Yaskawa INFORM job: A_ROOF_SIDE_0617_2_PAINT_35.JBI

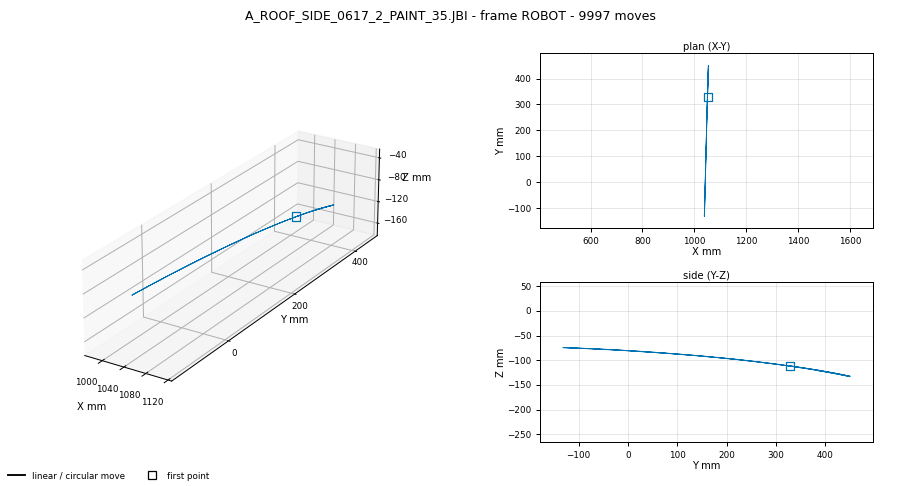
[picture p0: tool path of A_ROOF_SIDE_0617_2_PAINT_35.JBI in frame ROBOT, 9997 of 9997 moves have a stored position in this frame; points joined in program order, loops and branches not executed]
/JOB
//NAME A_ROOF_SIDE_0617_2_PAINT35
//POS
///NPOS 9997,0,0,0,0,0
///TOOL 1
///USER 0
///POSTYPE ROBOT
///RECTAN
///RCONF 1,0,0,0,0,0,0,0,0,0,0,0,0,0,0,0,0,0,0,0,0,0,0,0
C00000=1051.270,329.191,-111.247,172.986,38.897,157.407
C00001=1051.277,329.439,-111.283,172.990,38.901,157.408
C00002=1051.284,329.686,-111.318,172.994,38.904,157.409
C00003=1051.291,329.934,-111.353,172.998,38.908,157.410
C00004=1051.298,330.181,-111.388,173.002,38.912,157.411
C00005=1051.304,330.428,-111.423,173.006,38.916,157.412
C00006=1051.311,330.676,-111.458,173.010,38.920,157.414
C00007=1051.318,330.923,-111.494,173.014,38.924,157.414
C00008=1051.325,331.171,-111.529,173.018,38.928,157.415
C00009=1051.332,331.419,-111.564,173.022,38.933,157.417
C00010=1051.339,331.666,-111.599,173.026,38.936,157.418
C00011=1051.346,331.913,-111.635,173.031,38.940,157.419
C00012=1051.352,332.161,-111.670,173.035,38.944,157.420
C00013=1051.360,332.446,-111.711,173.039,38.949,157.421
C00014=1051.369,332.732,-111.752,173.044,38.953,157.422
C00015=1051.377,333.018,-111.792,173.049,38.958,157.423
C00016=1051.385,333.305,-111.834,173.054,38.963,157.424
C00017=1051.392,333.552,-111.869,173.058,38.967,157.426
C00018=1051.398,333.799,-111.904,173.062,38.971,157.427
C00019=1051.405,334.047,-111.940,173.066,38.975,157.428
C00020=1051.413,334.294,-111.976,173.070,38.979,157.429
C00021=1051.420,334.541,-112.011,173.075,38.983,157.430
C00022=1051.426,334.789,-112.046,173.079,38.988,157.431
C00023=1051.434,335.036,-112.082,173.083,38.991,157.432
C00024=1051.440,335.284,-112.118,173.087,38.996,157.433
C00025=1051.447,335.531,-112.153,173.092,39.000,157.434
C00026=1051.454,335.778,-112.189,173.096,39.003,157.435
C00027=1051.461,336.026,-112.225,173.100,39.008,157.436
C00028=1051.468,336.273,-112.260,173.104,39.012,157.437
C00029=1051.475,336.520,-112.296,173.109,39.016,157.438
C00030=1051.482,336.768,-112.332,173.113,39.021,157.439
C00031=1051.489,337.015,-112.367,173.117,39.024,157.440
C00032=1051.496,337.262,-112.403,173.122,39.029,157.441
C00033=1051.503,337.510,-112.439,173.126,39.033,157.442
C00034=1051.510,337.757,-112.475,173.130,39.037,157.444
C00035=1051.517,338.004,-112.511,173.134,39.041,157.445
C00036=1051.524,338.252,-112.547,173.139,39.045,157.446
C00037=1051.531,338.499,-112.583,173.143,39.050,157.447
C00038=1051.538,338.747,-112.619,173.147,39.054,157.448
C00039=1051.545,338.994,-112.654,173.152,39.058,157.449
C00040=1051.551,339.241,-112.691,173.156,39.062,157.450
C00041=1051.559,339.488,-112.727,173.160,39.067,157.451
C00042=1051.566,339.736,-112.762,173.165,39.071,157.452
C00043=1051.573,339.984,-112.799,173.169,39.075,157.453
C00044=1051.580,340.230,-112.835,173.173,39.079,157.455
C00045=1051.587,340.478,-112.872,173.178,39.084,157.456
C00046=1051.594,340.725,-112.908,173.182,39.088,157.457
C00047=1051.601,340.973,-112.943,173.186,39.092,157.458
C00048=1051.607,341.220,-112.979,173.191,39.096,157.459
C00049=1051.615,341.467,-113.016,173.195,39.101,157.460
C00050=1051.622,341.714,-113.052,173.199,39.105,157.461
C00051=1051.629,341.962,-113.088,173.204,39.109,157.462
C00052=1051.636,342.209,-113.124,173.209,39.114,157.464
C00053=1051.644,342.456,-113.160,173.213,39.117,157.465
C00054=1051.650,342.703,-113.197,173.218,39.122,157.466
C00055=1051.658,342.951,-113.233,173.222,39.126,157.467
C00056=1051.664,343.198,-113.270,173.227,39.131,157.468
C00057=1051.671,343.445,-113.306,173.231,39.135,157.469
C00058=1051.678,343.692,-113.342,173.235,39.139,157.470
C00059=1051.685,343.940,-113.379,173.240,39.144,157.471
C00060=1051.693,344.187,-113.416,173.244,39.148,157.473
C00061=1051.700,344.434,-113.452,173.249,39.152,157.474
C00062=1051.706,344.681,-113.489,173.253,39.157,157.475
C00063=1051.714,344.928,-113.525,173.258,39.162,157.476
C00064=1051.720,345.176,-113.562,173.262,39.166,157.477
C00065=1051.728,345.423,-113.599,173.266,39.170,157.478
C00066=1051.735,345.670,-113.635,173.272,39.175,157.480
C00067=1051.742,345.918,-113.672,173.276,39.179,157.481
C00068=1051.749,346.165,-113.708,173.281,39.183,157.482
C00069=1051.758,346.447,-113.751,173.286,39.189,157.483
C00070=1051.765,346.728,-113.792,173.291,39.194,157.485
C00071=1051.773,347.010,-113.834,173.296,39.199,157.486
C00072=1051.782,347.292,-113.876,173.301,39.204,157.487
C00073=1051.789,347.540,-113.913,173.306,39.209,157.489
C00074=1051.795,347.787,-113.950,173.310,39.213,157.490
C00075=1051.803,348.035,-113.987,173.315,39.218,157.491
C00076=1051.810,348.281,-114.023,173.319,39.222,157.492
C00077=1051.817,348.528,-114.061,173.324,39.227,157.493
C00078=1051.824,348.776,-114.098,173.328,39.231,157.494
C00079=1051.832,349.023,-114.135,173.334,39.236,157.496
C00080=1051.839,349.270,-114.172,173.338,39.240,157.497
C00081=1051.846,349.517,-114.209,173.343,39.245,157.498
C00082=1051.853,349.764,-114.246,173.348,39.249,157.499
C00083=1051.860,350.012,-114.282,173.352,39.254,157.500
C00084=1051.868,350.259,-114.320,173.357,39.259,157.502
C00085=1051.874,350.505,-114.357,173.361,39.263,157.503
C00086=1051.881,350.753,-114.394,173.367,39.268,157.504
C00087=1051.889,351.000,-114.431,173.371,39.272,157.505
C00088=1051.896,351.247,-114.468,173.376,39.277,157.507
C00089=1051.904,351.494,-114.506,173.380,39.281,157.508
C00090=1051.911,351.741,-114.543,173.385,39.286,157.509
C00091=1051.917,351.988,-114.580,173.389,39.291,157.510
C00092=1051.925,352.236,-114.617,173.395,39.296,157.512
C00093=1051.932,352.483,-114.655,173.400,39.300,157.513
C00094=1051.939,352.730,-114.692,173.404,39.305,157.514
C00095=1051.946,352.977,-114.730,173.409,39.310,157.515
C00096=1051.954,353.224,-114.767,173.414,39.315,157.517
C00097=1051.961,353.471,-114.805,173.419,39.319,157.518
C00098=1051.968,353.718,-114.842,173.424,39.324,157.519
C00099=1051.975,353.966,-114.880,173.428,39.329,157.520
C00100=1051.982,354.212,-114.917,173.433,39.333,157.522
C00101=1051.989,354.459,-114.955,173.437,39.338,157.523
C00102=1051.996,354.706,-114.992,173.443,39.343,157.524
C00103=1052.004,354.953,-115.030,173.448,39.348,157.525
C00104=1052.011,355.201,-115.067,173.452,39.352,157.527
C00105=1052.018,355.447,-115.106,173.457,39.357,157.528
C00106=1052.026,355.694,-115.143,173.463,39.362,157.529
C00107=1052.033,355.941,-115.181,173.467,39.366,157.531
C00108=1052.040,356.188,-115.218,173.472,39.371,157.532
C00109=1052.047,356.436,-115.256,173.477,39.376,157.533
C00110=1052.056,356.683,-115.294,173.482,39.381,157.534
C00111=1052.063,356.930,-115.332,173.487,39.386,157.536
C00112=1052.070,357.177,-115.369,173.492,39.391,157.537
C00113=1052.078,357.424,-115.408,173.496,39.396,157.538
C00114=1052.085,357.671,-115.445,173.502,39.401,157.540
C00115=1052.091,357.918,-115.483,173.507,39.405,157.541
C00116=1052.099,358.165,-115.521,173.511,39.410,157.542
C00117=1052.106,358.412,-115.559,173.516,39.415,157.544
C00118=1052.114,358.658,-115.597,173.522,39.420,157.545
C00119=1052.121,358.905,-115.635,173.527,39.425,157.546
C00120=1052.128,359.152,-115.674,173.531,39.430,157.548
C00121=1052.136,359.400,-115.711,173.537,39.435,157.549
C00122=1052.143,359.647,-115.750,173.542,39.440,157.550
C00123=1052.150,359.894,-115.787,173.546,39.445,157.552
C00124=1052.158,360.140,-115.825,173.551,39.450,157.553
C00125=1052.164,360.354,-115.859,173.555,39.454,157.554
C00126=1052.170,360.566,-115.892,173.561,39.458,157.555
C00127=1052.177,360.780,-115.924,173.565,39.463,157.556
C00128=1052.183,360.993,-115.957,173.569,39.467,157.558
C00129=1052.190,361.206,-115.990,173.573,39.471,157.559
C00130=1052.196,361.419,-116.024,173.578,39.476,157.560
C00131=1052.202,361.632,-116.057,173.582,39.480,157.561
C00132=1052.209,361.845,-116.090,173.587,39.485,157.562
C00133=1052.216,362.092,-116.128,173.592,39.489,157.564
C00134=1052.223,362.339,-116.167,173.597,39.495,157.565
C00135=1052.230,362.586,-116.205,173.603,39.500,157.567
C00136=1052.239,362.833,-116.243,173.607,39.505,157.568
C00137=1052.249,363.188,-116.298,173.615,39.512,157.570
C00138=1052.260,363.542,-116.354,173.622,39.520,157.572
C00139=1052.270,363.898,-116.410,173.630,39.527,157.574
C00140=1052.281,364.252,-116.465,173.637,39.534,157.576
C00141=1052.288,364.499,-116.504,173.642,39.539,157.577
C00142=1052.296,364.746,-116.543,173.647,39.545,157.579
C00143=1052.303,364.993,-116.582,173.653,39.550,157.580
C00144=1052.310,365.239,-116.620,173.658,39.555,157.582
C00145=1052.318,365.487,-116.659,173.664,39.560,157.583
C00146=1052.325,365.733,-116.698,173.669,39.566,157.585
C00147=1052.332,365.980,-116.737,173.674,39.571,157.586
C00148=1052.340,366.227,-116.776,173.679,39.576,157.587
C00149=1052.347,366.473,-116.815,173.684,39.581,157.589
C00150=1052.355,366.721,-116.854,173.690,39.587,157.590
C00151=1052.362,366.968,-116.892,173.695,39.592,157.592
C00152=1052.370,367.214,-116.932,173.701,39.597,157.593
C00153=1052.378,367.461,-116.970,173.706,39.603,157.595
C00154=1052.385,367.708,-117.009,173.711,39.608,157.596
C00155=1052.392,367.955,-117.049,173.717,39.613,157.598
C00156=1052.400,368.201,-117.087,173.722,39.619,157.599
C00157=1052.408,368.448,-117.127,173.728,39.624,157.601
C00158=1052.415,368.695,-117.165,173.732,39.630,157.602
C00159=1052.423,368.942,-117.205,173.738,39.635,157.603
C00160=1052.430,369.188,-117.244,173.743,39.640,157.605
C00161=1052.438,369.435,-117.284,173.749,39.646,157.606
C00162=1052.445,369.682,-117.323,173.754,39.651,157.608
C00163=1052.453,369.928,-117.362,173.760,39.656,157.609
C00164=1052.461,370.176,-117.401,173.765,39.662,157.611
C00165=1052.468,370.422,-117.440,173.770,39.667,157.612
C00166=1052.476,370.669,-117.480,173.776,39.673,157.614
C00167=1052.484,370.916,-117.519,173.782,39.678,157.615
C00168=1052.491,371.162,-117.559,173.787,39.684,157.617
C00169=1052.499,371.409,-117.598,173.792,39.689,157.618
C00170=1052.507,371.657,-117.637,173.798,39.695,157.620
C00171=1052.514,371.903,-117.677,173.804,39.700,157.621
C00172=1052.522,372.150,-117.717,173.809,39.705,157.623
C00173=1052.529,372.397,-117.756,173.816,39.711,157.625
C00174=1052.536,372.643,-117.796,173.821,39.716,157.626
C00175=1052.544,372.890,-117.836,173.827,39.722,157.628
C00176=1052.553,373.136,-117.875,173.832,39.728,157.629
C00177=1052.560,373.382,-117.915,173.838,39.734,157.631
C00178=1052.567,373.629,-117.955,173.843,39.739,157.632
C00179=1052.575,373.876,-117.995,173.849,39.745,157.634
C00180=1052.582,374.122,-118.034,173.855,39.751,157.635
C00181=1052.592,374.429,-118.084,173.861,39.758,157.637
C00182=1052.602,374.735,-118.133,173.868,39.765,157.639
C00183=1052.611,375.040,-118.183,173.875,39.772,157.641
C00184=1052.620,375.347,-118.233,173.882,39.779,157.643
C00185=1052.628,375.594,-118.272,173.888,39.785,157.645
C00186=1052.636,375.840,-118.313,173.895,39.791,157.647
C00187=1052.644,376.087,-118.353,173.900,39.796,157.648
C00188=1052.651,376.333,-118.392,173.906,39.802,157.650
C00189=1052.659,376.580,-118.432,173.911,39.808,157.651
C00190=1052.667,376.826,-118.473,173.917,39.813,157.653
C00191=1052.675,377.073,-118.513,173.923,39.819,157.655
C00192=1052.683,377.320,-118.553,173.929,39.825,157.656
C00193=1052.690,377.566,-118.593,173.935,39.831,157.658
C00194=1052.698,377.813,-118.633,173.941,39.837,157.659
C00195=1052.706,378.060,-118.674,173.946,39.843,157.661
C00196=1052.714,378.307,-118.714,173.952,39.848,157.663
C00197=1052.722,378.553,-118.754,173.959,39.854,157.664
C00198=1052.730,378.800,-118.794,173.964,39.860,157.666
C00199=1052.738,379.046,-118.835,173.970,39.866,157.668
C00200=1052.746,379.292,-118.875,173.976,39.872,157.669
C00201=1052.753,379.539,-118.915,173.981,39.878,157.671
C00202=1052.761,379.786,-118.956,173.988,39.884,157.673
C00203=1052.769,380.032,-118.996,173.994,39.890,157.674
C00204=1052.776,380.279,-119.037,173.999,39.896,157.676
C00205=1052.784,380.525,-119.078,174.005,39.902,157.678
C00206=1052.792,380.772,-119.118,174.012,39.908,157.679
C00207=1052.800,381.018,-119.160,174.018,39.914,157.681
C00208=1052.808,381.264,-119.200,174.023,39.920,157.683
C00209=1052.815,381.511,-119.240,174.030,39.926,157.685
C00210=1052.823,381.758,-119.281,174.036,39.932,157.686
C00211=1052.831,382.004,-119.322,174.042,39.938,157.688
C00212=1052.839,382.251,-119.363,174.047,39.944,157.690
C00213=1052.846,382.497,-119.404,174.054,39.951,157.692
C00214=1052.854,382.743,-119.445,174.060,39.957,157.693
C00215=1052.862,382.990,-119.485,174.066,39.963,157.695
C00216=1052.870,383.236,-119.527,174.072,39.969,157.697
C00217=1052.878,383.483,-119.568,174.078,39.975,157.699
C00218=1052.886,383.729,-119.609,174.084,39.981,157.700
C00219=1052.894,383.976,-119.650,174.091,39.988,157.702
C00220=1052.902,384.222,-119.691,174.097,39.994,157.704
C00221=1052.910,384.469,-119.732,174.104,40.000,157.706
C00222=1052.918,384.715,-119.774,174.109,40.007,157.707
C00223=1052.926,384.961,-119.814,174.115,40.013,157.709
C00224=1052.933,385.208,-119.855,174.122,40.019,157.711
C00225=1052.942,385.454,-119.897,174.128,40.025,157.713
C00226=1052.950,385.700,-119.938,174.135,40.031,157.714
C00227=1052.957,385.947,-119.979,174.140,40.038,157.716
C00228=1052.966,386.193,-120.021,174.147,40.044,157.718
C00229=1052.974,386.440,-120.062,174.153,40.051,157.720
C00230=1052.982,386.686,-120.103,174.159,40.057,157.722
C00231=1052.991,386.933,-120.144,174.166,40.063,157.724
C00232=1052.998,387.178,-120.186,174.172,40.070,157.725
C00233=1053.006,387.425,-120.227,174.179,40.076,157.727
C00234=1053.014,387.671,-120.269,174.185,40.082,157.729
C00235=1053.022,387.918,-120.310,174.192,40.089,157.731
C00236=1053.031,388.164,-120.352,174.198,40.096,157.733
C00237=1053.042,388.502,-120.409,174.207,40.104,157.735
C00238=1053.054,388.841,-120.466,174.216,40.113,157.738
C00239=1053.064,389.179,-120.523,174.224,40.122,157.741
C00240=1053.076,389.518,-120.580,174.233,40.131,157.743
C00241=1053.084,389.763,-120.622,174.240,40.137,157.745
C00242=1053.092,390.010,-120.664,174.246,40.144,157.747
C00243=1053.101,390.256,-120.706,174.253,40.151,157.749
C00244=1053.109,390.503,-120.748,174.260,40.157,157.751
C00245=1053.116,390.748,-120.790,174.266,40.164,157.753
C00246=1053.125,390.995,-120.832,174.273,40.171,157.755
C00247=1053.133,391.241,-120.874,174.279,40.178,157.757
C00248=1053.141,391.487,-120.916,174.286,40.184,157.758
C00249=1053.149,391.733,-120.957,174.293,40.191,157.760
C00250=1053.158,391.980,-120.999,174.299,40.198,157.762
C00251=1053.166,392.226,-121.043,174.306,40.204,157.764
C00252=1053.174,392.472,-121.084,174.313,40.211,157.766
C00253=1053.183,392.718,-121.126,174.319,40.218,157.768
C00254=1053.191,392.965,-121.168,174.326,40.225,157.770
C00255=1053.199,393.210,-121.211,174.333,40.232,157.772
C00256=1053.207,393.457,-121.253,174.340,40.238,157.774
C00257=1053.215,393.704,-121.296,174.347,40.245,157.776
C00258=1053.223,393.949,-121.338,174.354,40.252,157.778
C00259=1053.232,394.195,-121.380,174.360,40.259,157.780
C00260=1053.240,394.441,-121.423,174.367,40.266,157.782
C00261=1053.248,394.687,-121.465,174.374,40.273,157.784
C00262=1053.256,394.933,-121.508,174.380,40.280,157.786
C00263=1053.265,395.180,-121.550,174.387,40.287,157.788
C00264=1053.273,395.426,-121.593,174.394,40.294,157.790
C00265=1053.282,395.672,-121.636,174.402,40.301,157.792
C00266=1053.290,395.918,-121.678,174.408,40.308,157.794
C00267=1053.299,396.164,-121.721,174.415,40.315,157.796
C00268=1053.307,396.410,-121.764,174.422,40.322,157.798
C00269=1053.315,396.657,-121.806,174.429,40.329,157.801
C00270=1053.324,396.903,-121.849,174.436,40.336,157.803
C00271=1053.332,397.149,-121.892,174.443,40.343,157.805
C00272=1053.341,397.395,-121.935,174.450,40.351,157.807
C00273=1053.349,397.641,-121.978,174.457,40.358,157.809
C00274=1053.358,397.887,-122.021,174.464,40.364,157.811
C00275=1053.365,398.134,-122.064,174.472,40.372,157.813
C00276=1053.374,398.380,-122.107,174.479,40.379,157.815
C00277=1053.382,398.626,-122.150,174.485,40.386,157.817
C00278=1053.391,398.871,-122.194,174.492,40.394,157.820
C00279=1053.399,399.117,-122.237,174.500,40.401,157.822
C00280=1053.408,399.364,-122.280,174.507,40.408,157.824
C00281=1053.417,399.610,-122.323,174.514,40.415,157.826
C00282=1053.425,399.856,-122.366,174.522,40.423,157.828
C00283=1053.434,400.102,-122.409,174.529,40.430,157.830
C00284=1053.442,400.348,-122.452,174.536,40.438,157.833
C00285=1053.450,400.593,-122.497,174.544,40.445,157.835
C00286=1053.459,400.840,-122.540,174.551,40.452,157.837
C00287=1053.468,401.086,-122.583,174.558,40.459,157.839
C00288=1053.476,401.332,-122.627,174.566,40.467,157.841
C00289=1053.485,401.578,-122.670,174.573,40.474,157.843
C00290=1053.493,401.824,-122.713,174.581,40.482,157.846
C00291=1053.502,402.070,-122.757,174.588,40.489,157.848
C00292=1053.511,402.316,-122.800,174.595,40.497,157.850
C00293=1053.523,402.672,-122.864,174.606,40.508,157.853
C00294=1053.535,403.029,-122.927,174.616,40.519,157.857
C00295=1053.548,403.385,-122.991,174.627,40.530,157.860
C00296=1053.561,403.741,-123.054,174.638,40.541,157.863
C00297=1053.569,403.987,-123.097,174.646,40.549,157.866
C00298=1053.578,404.234,-123.142,174.653,40.557,157.868
C00299=1053.587,404.479,-123.186,174.661,40.564,157.870
C00300=1053.595,404.725,-123.231,174.668,40.572,157.873
C00301=1053.604,404.971,-123.274,174.676,40.580,157.875
C00302=1053.613,405.216,-123.318,174.683,40.588,157.877
C00303=1053.621,405.463,-123.363,174.692,40.595,157.880
C00304=1053.630,405.708,-123.407,174.699,40.603,157.882
C00305=1053.639,405.955,-123.451,174.707,40.611,157.884
C00306=1053.647,406.200,-123.496,174.715,40.619,157.887
C00307=1053.656,406.446,-123.540,174.722,40.627,157.889
C00308=1053.664,406.692,-123.584,174.730,40.634,157.891
C00309=1053.674,406.938,-123.628,174.738,40.643,157.894
C00310=1053.682,407.184,-123.672,174.746,40.650,157.896
C00311=1053.691,407.431,-123.717,174.754,40.659,157.899
C00312=1053.700,407.675,-123.762,174.761,40.666,157.901
C00313=1053.708,407.922,-123.806,174.770,40.674,157.903
C00314=1053.718,408.168,-123.850,174.778,40.683,157.906
C00315=1053.726,408.413,-123.895,174.785,40.690,157.908
C00316=1053.735,408.660,-123.940,174.793,40.699,157.911
C00317=1053.745,408.905,-123.985,174.802,40.707,157.913
C00318=1053.753,409.151,-124.029,174.809,40.715,157.916
C00319=1053.762,409.397,-124.075,174.817,40.723,157.918
C00320=1053.771,409.643,-124.119,174.826,40.731,157.921
C00321=1053.779,409.888,-124.164,174.833,40.740,157.923
C00322=1053.789,410.134,-124.208,174.841,40.748,157.926
C00323=1053.798,410.380,-124.253,174.850,40.756,157.928
C00324=1053.807,410.626,-124.299,174.858,40.764,157.931
C00325=1053.816,410.872,-124.343,174.866,40.772,157.933
C00326=1053.825,411.118,-124.388,174.874,40.781,157.936
C00327=1053.834,411.363,-124.433,174.883,40.789,157.938
C00328=1053.843,411.608,-124.478,174.891,40.797,157.941
C00329=1053.852,411.854,-124.524,174.900,40.805,157.943
C00330=1053.861,412.101,-124.568,174.907,40.814,157.946
C00331=1053.871,412.346,-124.613,174.915,40.822,157.948
C00332=1053.880,412.592,-124.659,174.924,40.831,157.951
C00333=1053.889,412.838,-124.704,174.933,40.839,157.954
C00334=1053.898,413.083,-124.749,174.941,40.847,157.956
C00335=1053.907,413.329,-124.794,174.950,40.856,157.959
C00336=1053.916,413.575,-124.840,174.958,40.865,157.961
C00337=1053.926,413.820,-124.886,174.967,40.873,157.964
C00338=1053.935,414.066,-124.931,174.975,40.882,157.967
C00339=1053.944,414.312,-124.977,174.984,40.891,157.969
C00340=1053.952,414.558,-125.022,174.992,40.899,157.972
C00341=1053.962,414.803,-125.068,175.000,40.908,157.975
C00342=1053.971,415.049,-125.114,175.009,40.917,157.977
C00343=1053.981,415.294,-125.160,175.017,40.925,157.980
C00344=1053.990,415.540,-125.206,175.026,40.934,157.983
C00345=1053.999,415.785,-125.252,175.035,40.942,157.985
C00346=1054.008,416.031,-125.297,175.044,40.952,157.988
C00347=1054.017,416.276,-125.343,175.053,40.960,157.991
C00348=1054.026,416.522,-125.389,175.062,40.969,157.994
C00349=1054.040,416.885,-125.458,175.074,40.982,157.998
C00350=1054.054,417.248,-125.525,175.088,40.995,158.002
C00351=1054.068,417.610,-125.593,175.100,41.008,158.006
C00352=1054.081,417.972,-125.661,175.114,41.021,158.010
C00353=1054.091,418.218,-125.708,175.123,41.031,158.013
C00354=1054.101,418.463,-125.754,175.132,41.040,158.016
C00355=1054.110,418.709,-125.800,175.141,41.049,158.019
C00356=1054.120,418.955,-125.846,175.150,41.058,158.021
C00357=1054.129,419.200,-125.892,175.159,41.067,158.024
C00358=1054.139,419.446,-125.939,175.168,41.076,158.027
C00359=1054.148,419.691,-125.985,175.177,41.085,158.030
C00360=1054.157,419.937,-126.032,175.187,41.094,158.033
C00361=1054.167,420.182,-126.079,175.196,41.104,158.036
C00362=1054.177,420.428,-126.126,175.205,41.113,158.039
C00363=1054.185,420.673,-126.172,175.215,41.122,158.042
C00364=1054.196,420.918,-126.219,175.224,41.131,158.045
C00365=1054.205,421.164,-126.266,175.233,41.141,158.048
C00366=1054.214,421.409,-126.313,175.243,41.150,158.050
C00367=1054.224,421.654,-126.360,175.252,41.160,158.053
C00368=1054.234,421.900,-126.407,175.261,41.169,158.056
C00369=1054.243,422.146,-126.454,175.271,41.178,158.059
C00370=1054.252,422.390,-126.501,175.280,41.188,158.062
C00371=1054.263,422.636,-126.548,175.290,41.197,158.065
C00372=1054.272,422.882,-126.595,175.299,41.207,158.068
C00373=1054.281,423.126,-126.642,175.308,41.216,158.071
C00374=1054.292,423.372,-126.689,175.319,41.226,158.074
C00375=1054.301,423.617,-126.737,175.328,41.235,158.078
C00376=1054.311,423.863,-126.783,175.338,41.246,158.081
C00377=1054.321,424.108,-126.830,175.347,41.255,158.084
C00378=1054.330,424.353,-126.878,175.357,41.265,158.087
C00379=1054.340,424.599,-126.925,175.368,41.274,158.090
C00380=1054.350,424.844,-126.973,175.377,41.284,158.093
C00381=1054.360,425.090,-127.020,175.387,41.294,158.096
C00382=1054.370,425.334,-127.068,175.397,41.303,158.099
C00383=1054.380,425.580,-127.116,175.407,41.313,158.103
C00384=1054.390,425.825,-127.163,175.417,41.324,158.106
C00385=1054.399,426.071,-127.211,175.427,41.333,158.109
C00386=1054.410,426.316,-127.258,175.437,41.343,158.112
C00387=1054.419,426.561,-127.307,175.447,41.353,158.115
C00388=1054.429,426.807,-127.355,175.457,41.363,158.118
C00389=1054.439,427.051,-127.403,175.467,41.373,158.122
C00390=1054.449,427.297,-127.450,175.477,41.383,158.125
C00391=1054.459,427.542,-127.498,175.488,41.393,158.128
C00392=1054.469,427.786,-127.547,175.497,41.403,158.131
C00393=1054.478,428.032,-127.595,175.508,41.414,158.135
C00394=1054.489,428.277,-127.643,175.518,41.424,158.138
C00395=1054.499,428.522,-127.691,175.529,41.433,158.141
C00396=1054.508,428.767,-127.739,175.539,41.444,158.145
C00397=1054.519,429.013,-127.787,175.550,41.454,158.148
C00398=1054.529,429.258,-127.836,175.560,41.464,158.151
C00399=1054.539,429.503,-127.884,175.570,41.475,158.155
C00400=1054.549,429.747,-127.932,175.581,41.485,158.158
C00401=1054.560,429.993,-127.981,175.591,41.496,158.161
C00402=1054.569,430.238,-128.030,175.602,41.506,158.165
C00403=1054.579,430.483,-128.078,175.613,41.516,158.168
C00404=1054.589,430.727,-128.127,175.623,41.527,158.172
C00405=1054.606,431.112,-128.204,175.641,41.543,158.177
C00406=1054.621,431.497,-128.280,175.657,41.560,158.183
C00407=1054.638,431.882,-128.357,175.674,41.577,158.188
C00408=1054.653,432.266,-128.434,175.692,41.593,158.194
C00409=1054.664,432.511,-128.483,175.703,41.604,158.197
C00410=1054.675,432.755,-128.532,175.713,41.615,158.201
C00411=1054.685,433.001,-128.581,175.724,41.625,158.204
C00412=1054.695,433.245,-128.630,175.735,41.636,158.208
C00413=1054.706,433.491,-128.680,175.747,41.647,158.211
C00414=1054.715,433.735,-128.728,175.758,41.658,158.215
C00415=1054.726,433.981,-128.778,175.769,41.669,158.219
C00416=1054.736,434.225,-128.827,175.780,41.680,158.222
C00417=1054.747,434.470,-128.877,175.792,41.691,158.226
C00418=1054.757,434.715,-128.926,175.803,41.702,158.230
C00419=1054.768,434.960,-128.976,175.814,41.713,158.233
C00420=1054.778,435.204,-129.025,175.826,41.724,158.237
C00421=1054.789,435.449,-129.075,175.837,41.735,158.241
C00422=1054.800,435.694,-129.125,175.849,41.746,158.244
C00423=1054.810,435.939,-129.175,175.860,41.757,158.248
C00424=1054.821,436.183,-129.224,175.873,41.768,158.252
C00425=1054.831,436.428,-129.273,175.884,41.780,158.256
C00426=1054.842,436.673,-129.324,175.896,41.791,158.260
C00427=1054.853,436.918,-129.373,175.907,41.802,158.263
C00428=1054.864,437.163,-129.423,175.919,41.814,158.267
C00429=1054.874,437.407,-129.473,175.931,41.825,158.271
C00430=1054.885,437.652,-129.524,175.943,41.836,158.275
C00431=1054.896,437.897,-129.573,175.954,41.848,158.279
C00432=1054.907,438.141,-129.624,175.967,41.859,158.283
C00433=1054.917,438.386,-129.675,175.979,41.870,158.286
C00434=1054.928,438.630,-129.725,175.990,41.882,158.290
C00435=1054.939,438.875,-129.775,176.003,41.894,158.294
C00436=1054.950,439.120,-129.825,176.015,41.905,158.298
C00437=1054.961,439.364,-129.875,176.028,41.917,158.302
C00438=1054.972,439.609,-129.927,176.039,41.929,158.306
C00439=1054.983,439.854,-129.977,176.052,41.940,158.310
C00440=1054.994,440.098,-130.028,176.064,41.953,158.314
C00441=1055.004,440.343,-130.079,176.077,41.964,158.318
C00442=1055.015,440.587,-130.129,176.089,41.976,158.322
C00443=1055.027,440.832,-130.180,176.102,41.988,158.326
C00444=1055.037,441.076,-130.231,176.114,42.000,158.331
C00445=1055.048,441.321,-130.282,176.126,42.011,158.335
C00446=1055.060,441.565,-130.333,176.140,42.023,158.339
C00447=1055.070,441.810,-130.384,176.152,42.036,158.343
C00448=1055.082,442.054,-130.435,176.165,42.048,158.347
C00449=1055.094,442.298,-130.486,176.178,42.060,158.351
C00450=1055.104,442.543,-130.537,176.191,42.072,158.355
C00451=1055.116,442.788,-130.589,176.203,42.084,158.360
C00452=1055.126,443.032,-130.640,176.216,42.096,158.364
C00453=1055.138,443.276,-130.692,176.229,42.109,158.368
C00454=1055.149,443.520,-130.743,176.242,42.121,158.372
C00455=1055.161,443.765,-130.795,176.256,42.133,158.377
C00456=1055.171,444.009,-130.846,176.269,42.146,158.381
C00457=1055.183,444.254,-130.898,176.282,42.158,158.385
C00458=1055.194,444.498,-130.949,176.295,42.170,158.390
C00459=1055.205,444.742,-131.001,176.309,42.183,158.394
C00460=1055.217,444.986,-131.054,176.322,42.196,158.399
C00461=1055.232,445.308,-131.121,176.339,42.212,158.404
C00462=1055.247,445.629,-131.189,176.357,42.229,158.410
C00463=1055.262,445.950,-131.257,176.376,42.245,158.416
C00464=1055.278,446.272,-131.326,176.393,42.262,158.422
C00465=1055.289,446.514,-131.378,176.406,42.275,158.426
C00466=1055.301,446.757,-131.430,176.421,42.287,158.431
C00467=1055.314,447.002,-131.481,176.434,42.300,158.435
C00468=1055.327,447.245,-131.532,176.449,42.312,158.440
C00469=1055.341,447.488,-131.582,176.462,42.324,158.444
C00470=1055.356,447.733,-131.632,176.476,42.336,158.448
C00471=1055.373,447.977,-131.681,176.491,42.348,158.453
C00472=1055.389,448.221,-131.729,176.505,42.359,158.457
C00473=1055.406,448.466,-131.777,176.519,42.371,158.461
C00474=1055.425,448.711,-131.824,176.533,42.382,158.465
C00475=1055.444,448.955,-131.870,176.548,42.393,158.469
C00476=1055.463,449.200,-131.917,176.562,42.404,158.473
C00477=1055.484,449.446,-131.962,176.577,42.414,158.477
C00478=1055.506,449.691,-132.007,176.592,42.425,158.481
C00479=1055.527,449.936,-132.051,176.606,42.435,158.485
C00480=1055.550,450.181,-132.095,176.621,42.445,158.489
C00481=1055.229,450.200,-132.384,176.619,42.547,158.518
C00482=1055.205,449.955,-132.340,176.604,42.538,158.514
C00483=1055.183,449.709,-132.297,176.589,42.527,158.510
C00484=1055.161,449.464,-132.252,176.574,42.517,158.506
C00485=1055.141,449.219,-132.206,176.559,42.506,158.502
C00486=1055.121,448.973,-132.160,176.545,42.496,158.498
C00487=1055.101,448.729,-132.114,176.530,42.485,158.494
C00488=1055.083,448.485,-132.066,176.516,42.474,158.490
C00489=1055.066,448.240,-132.018,176.502,42.462,158.486
C00490=1055.048,447.995,-131.971,176.488,42.451,158.482
C00491=1055.032,447.752,-131.922,176.474,42.439,158.477
C00492=1055.018,447.507,-131.872,176.459,42.428,158.473
C00493=1055.003,447.264,-131.823,176.445,42.415,158.469
C00494=1054.985,446.951,-131.757,176.427,42.400,158.463
C00495=1054.970,446.639,-131.691,176.409,42.384,158.457
C00496=1054.954,446.328,-131.625,176.392,42.368,158.451
C00497=1054.939,446.017,-131.558,176.374,42.352,158.446
C00498=1054.928,445.783,-131.509,176.360,42.340,158.441
C00499=1054.917,445.548,-131.459,176.348,42.328,158.437
C00500=1054.906,445.315,-131.409,176.335,42.316,158.433
C00501=1054.895,445.081,-131.359,176.322,42.303,158.429
C00502=1054.884,444.837,-131.307,176.308,42.291,158.424
C00503=1054.873,444.592,-131.255,176.295,42.279,158.420
C00504=1054.860,444.348,-131.203,176.281,42.266,158.415
C00505=1054.849,444.104,-131.152,176.268,42.254,158.411
C00506=1054.838,443.859,-131.100,176.255,42.242,158.407
C00507=1054.826,443.615,-131.049,176.242,42.229,158.403
C00508=1054.816,443.371,-130.997,176.228,42.217,158.398
C00509=1054.804,443.126,-130.946,176.215,42.205,158.394
C00510=1054.793,442.882,-130.894,176.202,42.193,158.390
C00511=1054.781,442.638,-130.843,176.190,42.180,158.385
C00512=1054.771,442.393,-130.791,176.177,42.168,158.381
C00513=1054.759,442.148,-130.740,176.163,42.156,158.377
C00514=1054.748,441.905,-130.689,176.150,42.144,158.373
C00515=1054.737,441.660,-130.637,176.137,42.132,158.369
C00516=1054.726,441.415,-130.587,176.125,42.121,158.365
C00517=1054.714,441.171,-130.536,176.112,42.109,158.360
C00518=1054.704,440.926,-130.485,176.099,42.097,158.356
C00519=1054.693,440.682,-130.434,176.087,42.085,158.352
C00520=1054.681,440.438,-130.383,176.074,42.073,158.348
C00521=1054.671,440.193,-130.333,176.062,42.061,158.344
C00522=1054.660,439.948,-130.282,176.050,42.050,158.340
C00523=1054.648,439.704,-130.231,176.038,42.037,158.336
C00524=1054.638,439.459,-130.180,176.025,42.026,158.332
C00525=1054.627,439.215,-130.130,176.013,42.014,158.328
C00526=1054.616,438.971,-130.079,176.000,42.003,158.324
C00527=1054.605,438.726,-130.029,175.989,41.992,158.320
C00528=1054.594,438.482,-129.979,175.976,41.980,158.316
C00529=1054.584,438.236,-129.928,175.964,41.968,158.312
C00530=1054.573,437.991,-129.878,175.951,41.957,158.308
C00531=1054.562,437.747,-129.827,175.940,41.945,158.304
C00532=1054.551,437.502,-129.777,175.928,41.934,158.301
C00533=1054.541,437.258,-129.728,175.916,41.923,158.297
C00534=1054.530,437.014,-129.677,175.904,41.911,158.293
C00535=1054.519,436.768,-129.628,175.892,41.900,158.289
C00536=1054.508,436.524,-129.578,175.881,41.889,158.285
C00537=1054.497,436.279,-129.528,175.869,41.878,158.281
C00538=1054.487,436.034,-129.478,175.857,41.867,158.278
C00539=1054.476,435.790,-129.428,175.845,41.856,158.274
C00540=1054.465,435.544,-129.378,175.834,41.845,158.270
C00541=1054.454,435.299,-129.329,175.822,41.834,158.267
C00542=1054.444,435.054,-129.279,175.811,41.823,158.263
C00543=1054.434,434.810,-129.230,175.799,41.812,158.259
C00544=1054.423,434.565,-129.180,175.788,41.800,158.255
C00545=1054.412,434.320,-129.131,175.777,41.790,158.252
C00546=1054.402,434.076,-129.081,175.765,41.779,158.248
C00547=1054.392,433.830,-129.032,175.754,41.768,158.245
C00548=1054.381,433.585,-128.982,175.743,41.757,158.241
C00549=1054.371,433.341,-128.933,175.732,41.747,158.237
C00550=1054.360,433.096,-128.883,175.720,41.736,158.234
C00551=1054.350,432.851,-128.835,175.709,41.725,158.230
C00552=1054.339,432.606,-128.786,175.698,41.714,158.227
C00553=1054.329,432.362,-128.737,175.686,41.703,158.223
C00554=1054.312,431.974,-128.660,175.669,41.687,158.217
C00555=1054.296,431.588,-128.582,175.652,41.670,158.212
C00556=1054.281,431.202,-128.504,175.635,41.654,158.206
C00557=1054.265,430.815,-128.428,175.617,41.637,158.201
C00558=1054.254,430.569,-128.379,175.607,41.626,158.197
C00559=1054.244,430.325,-128.330,175.596,41.616,158.194
C00560=1054.234,430.080,-128.281,175.585,41.606,158.191
C00561=1054.224,429.835,-128.233,175.575,41.595,158.187
C00562=1054.214,429.589,-128.184,175.564,41.585,158.184
C00563=1054.203,429.345,-128.136,175.553,41.575,158.180
C00564=1054.194,429.100,-128.088,175.544,41.565,158.177
C00565=1054.184,428.855,-128.039,175.533,41.554,158.174
C00566=1054.173,428.609,-127.991,175.522,41.544,158.170
C00567=1054.163,428.364,-127.943,175.512,41.534,158.167
C00568=1054.153,428.119,-127.894,175.501,41.524,158.164
C00569=1054.143,427.874,-127.846,175.491,41.514,158.160
C00570=1054.133,427.629,-127.798,175.480,41.504,158.157
C00571=1054.123,427.384,-127.751,175.471,41.494,158.154
C00572=1054.113,427.139,-127.702,175.460,41.484,158.151
C00573=1054.104,426.893,-127.654,175.450,41.474,158.147
C00574=1054.093,426.649,-127.606,175.440,41.464,158.144
C00575=1054.084,426.403,-127.559,175.430,41.454,158.141
C00576=1054.073,426.158,-127.511,175.420,41.444,158.138
C00577=1054.064,425.913,-127.463,175.409,41.434,158.135
C00578=1054.054,425.668,-127.416,175.399,41.424,158.131
C00579=1054.044,425.423,-127.367,175.390,41.415,158.128
C00580=1054.034,425.177,-127.320,175.379,41.405,158.125
C00581=1054.024,424.932,-127.272,175.369,41.395,158.122
C00582=1054.014,424.686,-127.225,175.360,41.385,158.119
C00583=1054.004,424.441,-127.178,175.349,41.376,158.116
C00584=1053.994,424.196,-127.130,175.340,41.366,158.113
C00585=1053.984,423.950,-127.083,175.330,41.356,158.109
C00586=1053.975,423.705,-127.035,175.321,41.347,158.106
C00587=1053.965,423.459,-126.988,175.311,41.337,158.103
C00588=1053.955,423.215,-126.941,175.300,41.328,158.100
C00589=1053.946,422.969,-126.894,175.291,41.318,158.097
C00590=1053.936,422.723,-126.847,175.281,41.309,158.094
C00591=1053.926,422.479,-126.800,175.272,41.299,158.091
C00592=1053.917,422.233,-126.752,175.262,41.290,158.088
C00593=1053.907,421.987,-126.705,175.253,41.281,158.085
C00594=1053.897,421.743,-126.658,175.244,41.271,158.082
C00595=1053.888,421.496,-126.611,175.234,41.261,158.079
C00596=1053.878,421.251,-126.564,175.225,41.252,158.076
C00597=1053.869,421.006,-126.518,175.215,41.243,158.073
C00598=1053.859,420.760,-126.470,175.205,41.234,158.070
C00599=1053.850,420.515,-126.424,175.196,41.224,158.067
C00600=1053.840,420.270,-126.377,175.187,41.215,158.064
C00601=1053.830,420.025,-126.331,175.178,41.206,158.062
C00602=1053.821,419.778,-126.284,175.169,41.197,158.059
C00603=1053.812,419.533,-126.238,175.159,41.188,158.056
C00604=1053.802,419.287,-126.191,175.150,41.179,158.053
C00605=1053.792,419.043,-126.144,175.141,41.169,158.050
C00606=1053.783,418.797,-126.098,175.132,41.160,158.047
C00607=1053.773,418.552,-126.052,175.122,41.151,158.044
C00608=1053.763,418.306,-126.005,175.113,41.143,158.042
C00609=1053.754,418.061,-125.959,175.104,41.134,158.039
C00610=1053.741,417.696,-125.891,175.091,41.121,158.035
C00611=1053.726,417.331,-125.822,175.078,41.107,158.030
C00612=1053.713,416.966,-125.754,175.064,41.094,158.026
C00613=1053.698,416.602,-125.685,175.052,41.081,158.022
C00614=1053.689,416.356,-125.640,175.042,41.072,158.019
C00615=1053.680,416.111,-125.593,175.033,41.063,158.017
C00616=1053.671,415.866,-125.547,175.025,41.055,158.014
C00617=1053.662,415.620,-125.502,175.016,41.046,158.011
C00618=1053.652,415.374,-125.455,175.007,41.037,158.008
C00619=1053.643,415.128,-125.410,174.999,41.028,158.006
C00620=1053.633,414.883,-125.364,174.990,41.020,158.003
C00621=1053.624,414.637,-125.318,174.981,41.011,158.000
C00622=1053.615,414.392,-125.273,174.973,41.003,157.998
C00623=1053.606,414.146,-125.227,174.964,40.994,157.995
C00624=1053.597,413.901,-125.181,174.955,40.985,157.992
C00625=1053.588,413.655,-125.136,174.947,40.977,157.990
C00626=1053.579,413.409,-125.090,174.938,40.969,157.987
C00627=1053.570,413.164,-125.045,174.930,40.960,157.984
C00628=1053.561,412.918,-124.999,174.921,40.951,157.982
C00629=1053.552,412.672,-124.954,174.913,40.943,157.979
C00630=1053.542,412.426,-124.909,174.904,40.934,157.977
C00631=1053.533,412.181,-124.863,174.897,40.926,157.974
C00632=1053.524,411.935,-124.818,174.888,40.918,157.972
C00633=1053.515,411.689,-124.773,174.880,40.909,157.969
C00634=1053.506,411.443,-124.728,174.871,40.901,157.966
C00635=1053.496,411.197,-124.684,174.863,40.893,157.964
C00636=1053.487,410.952,-124.638,174.854,40.885,157.961
C00637=1053.478,410.706,-124.593,174.847,40.877,157.959
C00638=1053.469,410.460,-124.548,174.838,40.869,157.956
C00639=1053.460,410.214,-124.503,174.830,40.860,157.954
C00640=1053.452,409.969,-124.458,174.821,40.852,157.951
C00641=1053.442,409.722,-124.414,174.814,40.844,157.949
C00642=1053.433,409.477,-124.369,174.806,40.836,157.946
C00643=1053.424,409.231,-124.323,174.797,40.828,157.944
C00644=1053.415,408.985,-124.280,174.789,40.820,157.941
C00645=1053.406,408.740,-124.234,174.781,40.811,157.939
C00646=1053.397,408.493,-124.190,174.773,40.804,157.936
C00647=1053.389,408.248,-124.146,174.765,40.796,157.934
C00648=1053.380,408.002,-124.100,174.757,40.787,157.932
C00649=1053.371,407.756,-124.056,174.749,40.780,157.929
C00650=1053.362,407.511,-124.011,174.741,40.771,157.927
C00651=1053.353,407.264,-123.967,174.733,40.764,157.924
C00652=1053.344,407.018,-123.922,174.726,40.755,157.922
C00653=1053.336,406.772,-123.878,174.718,40.748,157.920
C00654=1053.327,406.526,-123.834,174.710,40.740,157.917
C00655=1053.318,406.281,-123.789,174.702,40.732,157.915
C00656=1053.309,406.035,-123.745,174.694,40.724,157.912
C00657=1053.301,405.789,-123.700,174.687,40.716,157.910
C00658=1053.291,405.543,-123.656,174.679,40.709,157.908
C00659=1053.283,405.297,-123.612,174.671,40.701,157.905
C00660=1053.275,405.052,-123.568,174.663,40.693,157.903
C00661=1053.266,404.805,-123.523,174.655,40.685,157.901
C00662=1053.257,404.560,-123.480,174.648,40.677,157.898
C00663=1053.249,404.313,-123.436,174.640,40.670,157.896
C00664=1053.240,404.067,-123.392,174.633,40.662,157.894
C00665=1053.232,403.822,-123.348,174.625,40.655,157.891
C00666=1053.218,403.464,-123.284,174.614,40.643,157.888
C00667=1053.206,403.106,-123.220,174.603,40.633,157.885
C00668=1053.194,402.747,-123.156,174.593,40.621,157.881
C00669=1053.181,402.389,-123.092,174.581,40.610,157.878
C00670=1053.172,402.142,-123.049,174.574,40.603,157.876
C00671=1053.163,401.896,-123.005,174.566,40.595,157.874
C00672=1053.155,401.650,-122.962,174.559,40.588,157.871
C00673=1053.147,401.405,-122.918,174.551,40.580,157.869
C00674=1053.138,401.158,-122.874,174.544,40.573,157.867
C00675=1053.129,400.912,-122.831,174.537,40.566,157.865
C00676=1053.120,400.666,-122.788,174.529,40.559,157.863
C00677=1053.112,400.420,-122.745,174.522,40.551,157.860
C00678=1053.103,400.174,-122.702,174.514,40.544,157.858
C00679=1053.095,399.929,-122.657,174.507,40.536,157.856
C00680=1053.086,399.682,-122.614,174.500,40.529,157.854
C00681=1053.078,399.436,-122.571,174.492,40.522,157.852
C00682=1053.069,399.190,-122.528,174.486,40.515,157.850
C00683=1053.061,398.944,-122.485,174.479,40.507,157.847
C00684=1053.052,398.698,-122.442,174.472,40.500,157.845
C00685=1053.044,398.451,-122.399,174.464,40.493,157.843
C00686=1053.035,398.205,-122.356,174.457,40.486,157.841
C00687=1053.027,397.959,-122.313,174.450,40.479,157.839
C00688=1053.018,397.713,-122.270,174.442,40.472,157.837
C00689=1053.010,397.467,-122.227,174.435,40.464,157.835
C00690=1053.001,397.221,-122.184,174.429,40.457,157.833
C00691=1052.993,396.975,-122.140,174.422,40.450,157.831
C00692=1052.985,396.730,-122.097,174.414,40.443,157.828
C00693=1052.977,396.483,-122.054,174.407,40.436,157.826
C00694=1052.968,396.237,-122.013,174.400,40.429,157.824
C00695=1052.959,395.991,-121.970,174.394,40.422,157.822
C00696=1052.951,395.745,-121.927,174.387,40.415,157.820
C00697=1052.943,395.498,-121.884,174.380,40.408,157.818
C00698=1052.934,395.252,-121.841,174.372,40.401,157.816
C00699=1052.926,395.006,-121.798,174.366,40.394,157.814
C00700=1052.918,394.760,-121.756,174.359,40.387,157.812
C00701=1052.909,394.514,-121.714,174.352,40.380,157.810
C00702=1052.901,394.268,-121.671,174.345,40.373,157.808
C00703=1052.892,394.022,-121.628,174.339,40.367,157.806
C00704=1052.885,393.776,-121.586,174.331,40.360,157.804
C00705=1052.876,393.530,-121.543,174.324,40.353,157.802
C00706=1052.868,393.283,-121.501,174.317,40.346,157.800
C00707=1052.860,393.037,-121.459,174.311,40.339,157.798
C00708=1052.851,392.791,-121.417,174.304,40.333,157.796
C00709=1052.843,392.545,-121.374,174.297,40.326,157.794
C00710=1052.835,392.299,-121.333,174.291,40.319,157.792
C00711=1052.827,392.052,-121.290,174.284,40.312,157.790
C00712=1052.818,391.806,-121.248,174.277,40.306,157.788
C00713=1052.810,391.560,-121.206,174.271,40.299,157.786
C00714=1052.802,391.314,-121.164,174.263,40.292,157.784
C00715=1052.793,391.067,-121.122,174.258,40.286,157.782
C00716=1052.786,390.821,-121.080,174.250,40.279,157.780
C00717=1052.777,390.575,-121.038,174.243,40.272,157.778
C00718=1052.769,390.329,-120.996,174.237,40.266,157.776
C00719=1052.761,390.082,-120.954,174.230,40.259,157.775
C00720=1052.753,389.836,-120.912,174.224,40.253,157.773
C00721=1052.744,389.590,-120.870,174.217,40.246,157.771
C00722=1052.734,389.249,-120.812,174.209,40.237,157.768
C00723=1052.722,388.909,-120.755,174.199,40.228,157.766
C00724=1052.711,388.569,-120.698,174.190,40.219,157.763
C00725=1052.699,388.229,-120.640,174.182,40.210,157.760
C00726=1052.692,387.983,-120.599,174.175,40.204,157.759
C00727=1052.683,387.736,-120.557,174.169,40.197,157.757
C00728=1052.675,387.490,-120.516,174.162,40.191,157.755
C00729=1052.666,387.243,-120.474,174.156,40.185,157.753
C00730=1052.658,386.998,-120.433,174.149,40.178,157.751
C00731=1052.651,386.751,-120.391,174.143,40.172,157.749
C00732=1052.642,386.505,-120.350,174.136,40.166,157.748
C00733=1052.635,386.258,-120.309,174.130,40.159,157.746
C00734=1052.626,386.013,-120.267,174.123,40.153,157.744
C00735=1052.618,385.766,-120.226,174.118,40.147,157.742
C00736=1052.610,385.519,-120.185,174.112,40.140,157.740
C00737=1052.602,385.273,-120.144,174.105,40.134,157.738
C00738=1052.594,385.026,-120.102,174.099,40.128,157.737
C00739=1052.586,384.780,-120.061,174.092,40.122,157.735
C00740=1052.578,384.534,-120.020,174.086,40.115,157.733
C00741=1052.570,384.288,-119.979,174.079,40.109,157.731
C00742=1052.562,384.041,-119.938,174.074,40.103,157.730
C00743=1052.554,383.794,-119.897,174.068,40.097,157.728
C00744=1052.546,383.548,-119.855,174.061,40.091,157.726
C00745=1052.538,383.302,-119.815,174.055,40.085,157.724
C00746=1052.530,383.056,-119.774,174.049,40.078,157.723
C00747=1052.522,382.808,-119.732,174.042,40.072,157.721
C00748=1052.514,382.562,-119.692,174.037,40.066,157.719
C00749=1052.506,382.316,-119.651,174.031,40.060,157.717
C00750=1052.499,382.069,-119.610,174.024,40.054,157.715
C00751=1052.491,381.823,-119.569,174.018,40.048,157.714
C00752=1052.483,381.577,-119.529,174.012,40.041,157.712
C00753=1052.476,381.330,-119.487,174.006,40.036,157.710
C00754=1052.468,381.084,-119.447,174.000,40.030,157.709
C00755=1052.460,380.838,-119.406,173.994,40.023,157.707
C00756=1052.452,380.591,-119.365,173.988,40.018,157.705
C00757=1052.444,380.345,-119.324,173.982,40.011,157.703
C00758=1052.437,380.098,-119.284,173.976,40.006,157.702
C00759=1052.429,379.851,-119.244,173.970,40.000,157.700
C00760=1052.421,379.605,-119.202,173.965,39.994,157.699
C00761=1052.413,379.357,-119.162,173.958,39.988,157.697
C00762=1052.405,379.111,-119.121,173.952,39.982,157.695
C00763=1052.397,378.865,-119.081,173.946,39.976,157.693
C00764=1052.389,378.618,-119.041,173.941,39.970,157.692
C00765=1052.381,378.372,-119.000,173.934,39.964,157.690
C00766=1052.373,378.125,-118.960,173.928,39.958,157.688
C00767=1052.365,377.878,-118.920,173.923,39.953,157.687
C00768=1052.358,377.632,-118.880,173.917,39.947,157.685
C00769=1052.350,377.386,-118.840,173.910,39.941,157.684
C00770=1052.342,377.139,-118.800,173.905,39.935,157.682
C00771=1052.335,376.892,-118.760,173.899,39.930,157.680
C00772=1052.326,376.646,-118.720,173.893,39.924,157.679
C00773=1052.318,376.399,-118.680,173.888,39.918,157.677
C00774=1052.310,376.153,-118.639,173.882,39.912,157.675
C00775=1052.303,375.906,-118.599,173.875,39.907,157.674
C00776=1052.295,375.659,-118.559,173.870,39.901,157.672
C00777=1052.288,375.413,-118.520,173.864,39.895,157.671
C00778=1052.278,375.105,-118.469,173.857,39.888,157.669
C00779=1052.268,374.797,-118.419,173.850,39.881,157.667
C00780=1052.259,374.489,-118.369,173.843,39.874,157.665
C00781=1052.250,374.181,-118.319,173.836,39.867,157.663
C00782=1052.241,373.934,-118.280,173.831,39.861,157.661
C00783=1052.234,373.687,-118.240,173.824,39.856,157.660
C00784=1052.226,373.441,-118.201,173.818,39.850,157.658
C00785=1052.219,373.194,-118.161,173.813,39.844,157.656
C00786=1052.211,372.947,-118.121,173.807,39.839,157.655
C00787=1052.204,372.701,-118.081,173.802,39.833,157.653
C00788=1052.196,372.454,-118.041,173.796,39.828,157.652
C00789=1052.188,372.207,-118.001,173.791,39.822,157.650
C00790=1052.181,371.961,-117.962,173.785,39.817,157.649
C00791=1052.174,371.714,-117.922,173.780,39.811,157.647
C00792=1052.166,371.467,-117.882,173.774,39.805,157.646
C00793=1052.158,371.221,-117.844,173.768,39.800,157.644
C00794=1052.151,370.974,-117.804,173.763,39.795,157.643
C00795=1052.142,370.727,-117.765,173.757,39.789,157.641
C00796=1052.135,370.481,-117.726,173.752,39.784,157.640
C00797=1052.128,370.234,-117.686,173.746,39.778,157.638
C00798=1052.119,369.987,-117.646,173.741,39.773,157.637
C00799=1052.112,369.740,-117.608,173.735,39.768,157.635
C00800=1052.105,369.493,-117.568,173.730,39.762,157.634
C00801=1052.097,369.247,-117.529,173.724,39.757,157.632
C00802=1052.089,369.000,-117.490,173.719,39.752,157.631
C00803=1052.082,368.753,-117.451,173.713,39.746,157.629
C00804=1052.074,368.507,-117.411,173.708,39.741,157.628
C00805=1052.067,368.259,-117.372,173.702,39.736,157.626
C00806=1052.059,368.013,-117.333,173.697,39.730,157.625
C00807=1052.051,367.766,-117.294,173.692,39.725,157.623
C00808=1052.044,367.520,-117.255,173.686,39.720,157.622
C00809=1052.037,367.273,-117.216,173.681,39.714,157.620
C00810=1052.029,367.026,-117.178,173.675,39.709,157.619
C00811=1052.021,366.779,-117.138,173.670,39.704,157.617
C00812=1052.014,366.532,-117.099,173.665,39.699,157.616
C00813=1052.006,366.285,-117.061,173.660,39.693,157.615
C00814=1051.999,366.039,-117.021,173.654,39.688,157.613
C00815=1051.991,365.792,-116.982,173.649,39.683,157.612
C00816=1051.984,365.545,-116.944,173.644,39.678,157.610
C00817=1051.976,365.298,-116.905,173.638,39.672,157.609
C00818=1051.969,365.051,-116.866,173.633,39.667,157.607
C00819=1051.962,364.804,-116.827,173.627,39.662,157.606
C00820=1051.954,364.558,-116.788,173.623,39.657,157.605
C00821=1051.947,364.311,-116.749,173.617,39.652,157.603
C00822=1051.939,364.064,-116.711,173.612,39.647,157.602
C00823=1051.932,363.817,-116.672,173.607,39.641,157.600
C00824=1051.925,363.570,-116.633,173.601,39.637,157.599
C00825=1051.918,363.324,-116.595,173.596,39.631,157.597
C00826=1051.910,363.076,-116.556,173.592,39.626,157.596
C00827=1051.903,362.829,-116.517,173.586,39.621,157.595
C00828=1051.896,362.583,-116.479,173.581,39.616,157.593
C00829=1051.888,362.335,-116.441,173.575,39.611,157.592
C00830=1051.880,362.089,-116.403,173.570,39.606,157.591
C00831=1051.873,361.842,-116.364,173.565,39.601,157.589
C00832=1051.865,361.595,-116.325,173.560,39.596,157.588
C00833=1051.858,361.348,-116.287,173.555,39.591,157.586
C00834=1051.850,361.059,-116.242,173.549,39.585,157.585
C00835=1051.841,360.770,-116.198,173.543,39.579,157.583
C00836=1051.832,360.481,-116.152,173.537,39.573,157.582
C00837=1051.823,360.192,-116.108,173.531,39.568,157.580
C00838=1051.816,359.945,-116.070,173.526,39.562,157.579
C00839=1051.809,359.698,-116.032,173.521,39.558,157.577
C00840=1051.801,359.451,-115.993,173.516,39.553,157.576
C00841=1051.794,359.204,-115.956,173.511,39.548,157.575
C00842=1051.786,358.957,-115.918,173.506,39.543,157.573
C00843=1051.780,358.710,-115.879,173.501,39.538,157.572
C00844=1051.772,358.463,-115.841,173.496,39.533,157.571
C00845=1051.765,358.216,-115.804,173.491,39.529,157.569
C00846=1051.757,357.969,-115.765,173.486,39.524,157.568
C00847=1051.750,357.722,-115.728,173.481,39.519,157.567
C00848=1051.743,357.475,-115.689,173.476,39.514,157.566
C00849=1051.736,357.228,-115.651,173.471,39.509,157.564
C00850=1051.728,356.981,-115.614,173.466,39.504,157.563
C00851=1051.721,356.734,-115.575,173.461,39.499,157.562
C00852=1051.713,356.487,-115.538,173.456,39.495,157.560
C00853=1051.706,356.240,-115.500,173.451,39.490,157.559
C00854=1051.699,355.993,-115.463,173.446,39.485,157.558
C00855=1051.691,355.746,-115.425,173.441,39.480,157.556
C00856=1051.684,355.499,-115.387,173.437,39.476,157.555
C00857=1051.677,355.252,-115.350,173.431,39.471,157.554
C00858=1051.670,355.005,-115.312,173.427,39.466,157.553
C00859=1051.662,354.758,-115.275,173.422,39.461,157.551
C00860=1051.655,354.510,-115.237,173.417,39.456,157.550
C00861=1051.648,354.263,-115.199,173.412,39.452,157.549
C00862=1051.641,354.016,-115.162,173.407,39.447,157.547
C00863=1051.633,353.769,-115.124,173.402,39.442,157.546
C00864=1051.626,353.522,-115.087,173.398,39.438,157.545
C00865=1051.619,353.275,-115.049,173.392,39.433,157.544
C00866=1051.612,353.028,-115.012,173.388,39.428,157.542
C00867=1051.605,352.780,-114.974,173.383,39.424,157.541
C00868=1051.598,352.534,-114.937,173.378,39.419,157.540
C00869=1051.591,352.287,-114.900,173.374,39.414,157.539
C00870=1051.583,352.040,-114.862,173.368,39.410,157.537
C00871=1051.576,351.793,-114.825,173.364,39.405,157.536
C00872=1051.568,351.546,-114.788,173.359,39.400,157.535
C00873=1051.561,351.299,-114.750,173.355,39.396,157.534
C00874=1051.554,351.052,-114.713,173.350,39.391,157.533
C00875=1051.547,350.805,-114.676,173.344,39.386,157.531
C00876=1051.540,350.557,-114.639,173.340,39.382,157.530
C00877=1051.533,350.310,-114.601,173.335,39.377,157.529
C00878=1051.525,350.063,-114.565,173.331,39.373,157.528
C00879=1051.518,349.816,-114.527,173.326,39.368,157.526
C00880=1051.511,349.569,-114.490,173.322,39.364,157.525
C00881=1051.504,349.321,-114.453,173.317,39.359,157.524
C00882=1051.496,349.075,-114.416,173.312,39.355,157.523
C00883=1051.489,348.827,-114.380,173.307,39.350,157.521
C00884=1051.482,348.580,-114.342,173.303,39.346,157.520
C00885=1051.475,348.333,-114.305,173.298,39.341,157.519
C00886=1051.468,348.086,-114.269,173.294,39.337,157.518
C00887=1051.461,347.839,-114.231,173.289,39.332,157.517
C00888=1051.454,347.591,-114.194,173.284,39.328,157.516
C00889=1051.446,347.344,-114.157,173.279,39.323,157.514
C00890=1051.438,347.060,-114.116,173.274,39.318,157.513
C00891=1051.430,346.777,-114.073,173.269,39.313,157.512
C00892=1051.422,346.493,-114.030,173.264,39.308,157.510
C00893=1051.414,346.209,-113.989,173.258,39.303,157.509
C00894=1051.407,345.961,-113.952,173.254,39.298,157.508
C00895=1051.400,345.715,-113.915,173.249,39.294,157.507
C00896=1051.392,345.467,-113.879,173.245,39.290,157.505
C00897=1051.385,345.219,-113.842,173.240,39.285,157.504
C00898=1051.378,344.973,-113.805,173.236,39.281,157.503
C00899=1051.371,344.726,-113.769,173.232,39.277,157.502
C00900=1051.364,344.478,-113.732,173.226,39.272,157.501
C00901=1051.357,344.231,-113.696,173.222,39.268,157.500
C00902=1051.349,343.929,-113.651,173.217,39.262,157.498
C00903=1051.340,343.627,-113.607,173.211,39.257,157.497
C00904=1051.331,343.324,-113.562,173.205,39.252,157.495
C00905=1051.323,343.022,-113.517,173.200,39.247,157.494
C00906=1051.316,342.775,-113.481,173.196,39.242,157.493
C00907=1051.309,342.527,-113.444,173.191,39.238,157.492
C00908=1051.302,342.281,-113.408,173.187,39.234,157.491
C00909=1051.295,342.033,-113.371,173.183,39.229,157.489
C00910=1051.288,341.786,-113.336,173.178,39.225,157.488
C00911=1051.280,341.539,-113.299,173.174,39.221,157.487
C00912=1051.273,341.291,-113.263,173.169,39.217,157.486
C00913=1051.266,341.044,-113.227,173.165,39.212,157.485
C00914=1051.259,340.796,-113.191,173.160,39.208,157.484
C00915=1051.252,340.549,-113.155,173.156,39.204,157.483
C00916=1051.245,340.302,-113.119,173.151,39.200,157.482
C00917=1051.238,340.055,-113.083,173.147,39.195,157.481
C00918=1051.231,339.808,-113.046,173.142,39.191,157.479
C00919=1051.224,339.560,-113.011,173.138,39.187,157.478
C00920=1051.217,339.313,-112.975,173.134,39.183,157.477
C00921=1051.210,339.065,-112.938,173.129,39.178,157.476
C00922=1051.203,338.819,-112.902,173.125,39.175,157.475
C00923=1051.195,338.570,-112.867,173.121,39.170,157.474
C00924=1051.189,338.323,-112.830,173.116,39.166,157.473
C00925=1051.182,338.077,-112.794,173.112,39.162,157.472
C00926=1051.175,337.829,-112.759,173.108,39.158,157.471
C00927=1051.168,337.582,-112.722,173.104,39.154,157.470
C00928=1051.161,337.334,-112.686,173.099,39.149,157.469
C00929=1051.154,337.087,-112.651,173.095,39.145,157.467
C00930=1051.147,336.840,-112.615,173.091,39.141,157.466
C00931=1051.140,336.592,-112.579,173.086,39.137,157.465
C00932=1051.133,336.345,-112.543,173.082,39.133,157.464
C00933=1051.127,336.097,-112.508,173.078,39.128,157.463
C00934=1051.119,335.850,-112.471,173.074,39.125,157.462
C00935=1051.113,335.602,-112.436,173.069,39.120,157.461
C00936=1051.105,335.356,-112.400,173.065,39.116,157.460
C00937=1051.098,335.108,-112.365,173.061,39.113,157.459
C00938=1051.091,334.860,-112.330,173.057,39.108,157.458
C00939=1051.084,334.613,-112.294,173.052,39.104,157.457
C00940=1051.077,334.366,-112.259,173.048,39.101,157.456
C00941=1051.070,334.118,-112.223,173.044,39.096,157.455
C00942=1051.063,333.878,-112.189,173.040,39.092,157.454
C00943=1051.057,333.638,-112.154,173.036,39.088,157.453
C00944=1051.050,333.399,-112.120,173.031,39.085,157.452
C00945=1051.043,333.158,-112.085,173.027,39.081,157.451
C00946=1051.037,332.918,-112.051,173.024,39.077,157.450
C00947=1051.030,332.678,-112.016,173.020,39.073,157.449
C00948=1051.023,332.438,-111.982,173.016,39.069,157.448
C00949=1051.016,332.198,-111.948,173.012,39.065,157.447
C00950=1051.009,331.951,-111.913,173.008,39.061,157.446
C00951=1051.003,331.703,-111.877,173.004,39.057,157.445
C00952=1050.996,331.456,-111.842,172.999,39.053,157.444
C00953=1050.989,331.208,-111.806,172.995,39.049,157.442
C00954=1050.982,330.960,-111.771,172.991,39.045,157.441
C00955=1050.975,330.713,-111.736,172.987,39.041,157.440
C00956=1050.969,330.465,-111.701,172.983,39.037,157.439
C00957=1050.962,330.218,-111.666,172.979,39.033,157.438
C00958=1050.955,329.971,-111.631,172.974,39.029,157.437
C00959=1050.948,329.723,-111.595,172.970,39.025,157.436
C00960=1050.940,329.476,-111.561,172.966,39.021,157.435
C00961=1050.933,329.228,-111.525,172.962,39.017,157.434
C00962=1050.927,328.981,-111.490,172.958,39.014,157.433
C00963=1050.919,328.734,-111.456,172.955,39.010,157.432
C00964=1050.912,328.486,-111.421,172.950,39.006,157.431
C00965=1050.906,328.239,-111.386,172.946,39.002,157.430
C00966=1050.898,327.991,-111.352,172.942,38.999,157.429
C00967=1050.891,327.743,-111.316,172.938,38.995,157.428
C00968=1050.884,327.496,-111.281,172.934,38.991,157.427
C00969=1050.877,327.249,-111.246,172.930,38.987,157.427
C00970=1050.870,327.001,-111.212,172.926,38.983,157.426
C00971=1050.864,326.754,-111.177,172.921,38.980,157.425
C00972=1050.856,326.507,-111.142,172.917,38.976,157.424
C00973=1050.850,326.259,-111.108,172.914,38.972,157.423
C00974=1050.842,326.012,-111.073,172.910,38.968,157.422
C00975=1050.835,325.764,-111.038,172.906,38.964,157.421
C00976=1050.829,325.516,-111.004,172.902,38.961,157.420
C00977=1050.821,325.269,-110.969,172.898,38.957,157.419
C00978=1050.815,325.021,-110.935,172.894,38.953,157.418
C00979=1050.807,324.774,-110.900,172.890,38.949,157.417
C00980=1050.801,324.527,-110.865,172.886,38.945,157.416
C00981=1050.794,324.279,-110.831,172.882,38.941,157.415
C00982=1050.787,324.032,-110.796,172.878,38.938,157.414
C00983=1050.780,323.784,-110.762,172.874,38.934,157.413
C00984=1050.773,323.536,-110.727,172.870,38.930,157.412
C00985=1050.766,323.289,-110.693,172.866,38.926,157.411
C00986=1050.759,323.041,-110.658,172.862,38.923,157.410
C00987=1050.752,322.794,-110.624,172.858,38.919,157.409
C00988=1050.746,322.546,-110.590,172.854,38.915,157.408
C00989=1050.738,322.299,-110.555,172.850,38.912,157.407
C00990=1050.732,322.051,-110.521,172.847,38.908,157.406
C00991=1050.726,321.804,-110.486,172.843,38.904,157.405
C00992=1050.718,321.556,-110.452,172.839,38.900,157.404
C00993=1050.712,321.308,-110.418,172.835,38.897,157.403
C00994=1050.705,321.061,-110.383,172.831,38.893,157.402
C00995=1050.698,320.813,-110.349,172.827,38.889,157.401
C00996=1050.691,320.566,-110.315,172.823,38.885,157.400
C00997=1050.685,320.318,-110.281,172.820,38.882,157.400
C00998=1050.678,320.071,-110.246,172.816,38.878,157.399
C00999=1050.671,319.823,-110.212,172.812,38.874,157.398
C01000=1050.665,319.575,-110.177,172.808,38.870,157.397
C01001=1050.657,319.328,-110.144,172.804,38.867,157.396
C01002=1050.650,319.035,-110.103,172.800,38.863,157.395
C01003=1050.642,318.742,-110.062,172.795,38.858,157.394
C01004=1050.634,318.449,-110.022,172.791,38.854,157.392
C01005=1050.626,318.156,-109.981,172.786,38.849,157.391
C01006=1050.619,317.909,-109.947,172.782,38.846,157.390
C01007=1050.613,317.661,-109.913,172.779,38.842,157.390
C01008=1050.606,317.414,-109.879,172.775,38.839,157.389
C01009=1050.599,317.166,-109.845,172.771,38.835,157.388
C01010=1050.592,316.919,-109.812,172.767,38.831,157.387
C01011=1050.586,316.671,-109.777,172.764,38.828,157.386
C01012=1050.579,316.423,-109.743,172.760,38.824,157.385
C01013=1050.573,316.176,-109.709,172.757,38.820,157.384
C01014=1050.566,315.928,-109.675,172.753,38.817,157.383
C01015=1050.559,315.680,-109.641,172.749,38.813,157.382
C01016=1050.553,315.433,-109.608,172.745,38.809,157.381
C01017=1050.546,315.185,-109.573,172.741,38.805,157.380
C01018=1050.540,314.938,-109.540,172.737,38.802,157.379
C01019=1050.533,314.690,-109.505,172.734,38.798,157.378
C01020=1050.526,314.443,-109.471,172.730,38.795,157.378
C01021=1050.520,314.195,-109.437,172.727,38.791,157.377
C01022=1050.513,313.947,-109.404,172.723,38.788,157.376
C01023=1050.507,313.700,-109.370,172.719,38.784,157.375
C01024=1050.500,313.452,-109.336,172.716,38.780,157.374
C01025=1050.494,313.205,-109.302,172.712,38.776,157.373
C01026=1050.487,312.957,-109.269,172.708,38.773,157.372
C01027=1050.480,312.709,-109.235,172.704,38.770,157.371
C01028=1050.474,312.462,-109.202,172.700,38.766,157.370
C01029=1050.466,312.214,-109.168,172.698,38.762,157.369
C01030=1050.460,311.966,-109.135,172.694,38.759,157.369
C01031=1050.453,311.719,-109.102,172.690,38.756,157.368
C01032=1050.446,311.471,-109.068,172.686,38.752,157.367
C01033=1050.439,311.224,-109.035,172.682,38.749,157.366
C01034=1050.432,310.976,-109.001,172.679,38.745,157.365
C01035=1050.425,310.728,-108.968,172.675,38.742,157.364
C01036=1050.419,310.481,-108.935,172.671,38.739,157.363
C01037=1050.412,310.232,-108.902,172.669,38.735,157.363
C01038=1050.404,309.986,-108.869,172.665,38.731,157.362
C01039=1050.398,309.738,-108.836,172.661,38.728,157.361
C01040=1050.391,309.491,-108.802,172.657,38.725,157.360
C01041=1050.384,309.242,-108.769,172.653,38.721,157.359
C01042=1050.378,308.995,-108.736,172.650,38.718,157.358
C01043=1050.371,308.747,-108.702,172.646,38.715,157.357
C01044=1050.364,308.499,-108.670,172.643,38.711,157.356
C01045=1050.357,308.252,-108.636,172.639,38.707,157.356
C01046=1050.351,308.004,-108.603,172.636,38.704,157.355
C01047=1050.344,307.756,-108.570,172.632,38.701,157.354
C01048=1050.337,307.509,-108.537,172.628,38.697,157.353
C01049=1050.330,307.261,-108.504,172.624,38.694,157.352
C01050=1050.323,307.013,-108.471,172.622,38.690,157.351
C01051=1050.317,306.766,-108.438,172.618,38.687,157.351
C01052=1050.310,306.518,-108.405,172.614,38.683,157.350
C01053=1050.304,306.270,-108.372,172.610,38.680,157.349
C01054=1050.296,306.023,-108.338,172.607,38.676,157.348
C01055=1050.290,305.775,-108.305,172.604,38.673,157.347
C01056=1050.284,305.528,-108.273,172.600,38.670,157.346
C01057=1050.276,305.280,-108.240,172.596,38.666,157.345
C01058=1050.269,304.991,-108.201,172.592,38.662,157.345
C01059=1050.261,304.703,-108.163,172.589,38.659,157.344
C01060=1050.253,304.414,-108.124,172.584,38.655,157.343
C01061=1050.246,304.126,-108.087,172.580,38.651,157.342
C01062=1050.239,303.878,-108.054,172.577,38.647,157.341
C01063=1050.232,303.630,-108.021,172.573,38.644,157.340
C01064=1050.226,303.383,-107.987,172.570,38.641,157.339
C01065=1050.219,303.135,-107.955,172.566,38.637,157.338
C01066=1050.212,302.887,-107.922,172.563,38.634,157.337
C01067=1050.206,302.639,-107.889,172.560,38.630,157.337
C01068=1050.199,302.392,-107.857,172.556,38.627,157.336
C01069=1050.193,302.144,-107.824,172.552,38.623,157.335
C01070=1050.186,301.896,-107.791,172.549,38.620,157.334
C01071=1050.179,301.649,-107.759,172.545,38.616,157.333
C01072=1050.173,301.401,-107.726,172.542,38.613,157.332
C01073=1050.166,301.154,-107.693,172.539,38.610,157.331
C01074=1050.160,300.905,-107.660,172.535,38.606,157.331
C01075=1050.153,300.658,-107.627,172.532,38.603,157.330
C01076=1050.147,300.410,-107.595,172.529,38.599,157.329
C01077=1050.140,300.162,-107.563,172.525,38.596,157.328
C01078=1050.134,299.915,-107.530,172.521,38.593,157.327
C01079=1050.127,299.666,-107.497,172.519,38.589,157.326
C01080=1050.121,299.419,-107.465,172.515,38.586,157.326
C01081=1050.114,299.171,-107.432,172.511,38.583,157.325
C01082=1050.107,298.924,-107.400,172.509,38.579,157.324
C01083=1050.101,298.676,-107.367,172.505,38.576,157.323
C01084=1050.095,298.428,-107.335,172.501,38.573,157.322
C01085=1050.089,298.180,-107.302,172.498,38.570,157.322
C01086=1050.082,297.932,-107.269,172.495,38.566,157.321
C01087=1050.075,297.685,-107.237,172.491,38.563,157.320
C01088=1050.069,297.437,-107.205,172.488,38.559,157.319
C01089=1050.063,297.189,-107.172,172.485,38.556,157.318
C01090=1050.056,296.941,-107.139,172.481,38.553,157.318
C01091=1050.050,296.694,-107.108,172.478,38.549,157.317
C01092=1050.043,296.446,-107.075,172.474,38.546,157.316
C01093=1050.037,296.198,-107.043,172.472,38.543,157.315
C01094=1050.031,295.950,-107.010,172.468,38.539,157.314
C01095=1050.023,295.702,-106.978,172.464,38.536,157.313
C01096=1050.017,295.455,-106.945,172.462,38.533,157.313
C01097=1050.010,295.207,-106.914,172.458,38.530,157.312
C01098=1050.004,294.959,-106.881,172.454,38.526,157.311
C01099=1049.997,294.711,-106.850,172.452,38.523,157.310
C01100=1049.990,294.464,-106.817,172.448,38.520,157.310
C01101=1049.984,294.216,-106.785,172.445,38.517,157.309
C01102=1049.978,293.968,-106.754,172.442,38.513,157.308
C01103=1049.971,293.720,-106.721,172.438,38.510,157.307
C01104=1049.965,293.472,-106.690,172.435,38.507,157.306
C01105=1049.957,293.224,-106.657,172.432,38.504,157.306
C01106=1049.951,292.976,-106.625,172.429,38.500,157.305
C01107=1049.944,292.728,-106.594,172.425,38.497,157.304
C01108=1049.938,292.481,-106.561,172.421,38.494,157.303
C01109=1049.931,292.233,-106.530,172.419,38.491,157.302
C01110=1049.925,291.985,-106.498,172.415,38.487,157.302
C01111=1049.918,291.737,-106.466,172.412,38.484,157.301
C01112=1049.912,291.489,-106.434,172.409,38.481,157.300
C01113=1049.905,291.241,-106.403,172.406,38.478,157.299
C01114=1049.898,290.969,-106.367,172.402,38.474,157.298
C01115=1049.890,290.697,-106.332,172.399,38.471,157.298
C01116=1049.884,290.424,-106.297,172.395,38.467,157.297
C01117=1049.876,290.152,-106.263,172.391,38.463,157.296
C01118=1049.870,289.904,-106.230,172.389,38.461,157.295
C01119=1049.863,289.656,-106.199,172.385,38.457,157.294
C01120=1049.856,289.408,-106.167,172.382,38.454,157.293
C01121=1049.850,289.160,-106.136,172.379,38.451,157.293
C01122=1049.844,288.912,-106.104,172.376,38.447,157.292
C01123=1049.837,288.664,-106.072,172.372,38.445,157.291
C01124=1049.830,288.416,-106.041,172.370,38.441,157.290
C01125=1049.823,288.169,-106.009,172.366,38.438,157.290
C01126=1049.817,287.921,-105.977,172.363,38.435,157.289
C01127=1049.811,287.673,-105.945,172.360,38.432,157.288
C01128=1049.804,287.425,-105.914,172.357,38.428,157.287
C01129=1049.797,287.177,-105.883,172.353,38.425,157.287
C01130=1049.790,286.929,-105.851,172.350,38.422,157.286
C01131=1049.784,286.681,-105.820,172.347,38.419,157.285
C01132=1049.777,286.433,-105.788,172.343,38.416,157.284
C01133=1049.771,286.186,-105.758,172.341,38.413,157.284
C01134=1049.764,285.938,-105.726,172.337,38.409,157.283
C01135=1049.758,285.690,-105.695,172.334,38.407,157.282
C01136=1049.751,285.442,-105.664,172.331,38.403,157.281
C01137=1049.744,285.194,-105.632,172.328,38.400,157.281
C01138=1049.737,284.946,-105.601,172.324,38.397,157.280
C01139=1049.731,284.698,-105.569,172.322,38.394,157.279
C01140=1049.725,284.450,-105.537,172.319,38.391,157.278
C01141=1049.718,284.201,-105.507,172.316,38.388,157.278
C01142=1049.712,283.954,-105.475,172.313,38.384,157.277
C01143=1049.705,283.706,-105.444,172.309,38.382,157.276
C01144=1049.699,283.458,-105.413,172.307,38.378,157.275
C01145=1049.692,283.211,-105.381,172.303,38.375,157.275
C01146=1049.686,282.962,-105.350,172.300,38.372,157.274
C01147=1049.679,282.714,-105.319,172.297,38.369,157.273
C01148=1049.673,282.467,-105.288,172.294,38.366,157.272
C01149=1049.666,282.219,-105.257,172.291,38.363,157.272
C01150=1049.660,281.970,-105.226,172.288,38.359,157.271
C01151=1049.653,281.723,-105.194,172.285,38.356,157.270
C01152=1049.646,281.475,-105.163,172.282,38.353,157.269
C01153=1049.640,281.227,-105.133,172.279,38.350,157.269
C01154=1049.634,280.979,-105.101,172.275,38.347,157.268
C01155=1049.627,280.731,-105.070,172.273,38.344,157.267
C01156=1049.621,280.483,-105.039,172.269,38.341,157.266
C01157=1049.614,280.235,-105.008,172.266,38.338,157.266
C01158=1049.608,279.987,-104.977,172.264,38.334,157.265
C01159=1049.601,279.739,-104.946,172.260,38.331,157.264
C01160=1049.595,279.491,-104.914,172.258,38.328,157.263
C01161=1049.589,279.243,-104.884,172.254,38.325,157.263
C01162=1049.582,278.995,-104.853,172.251,38.322,157.262
C01163=1049.575,278.747,-104.822,172.249,38.319,157.261
C01164=1049.568,278.499,-104.791,172.245,38.316,157.260
C01165=1049.562,278.251,-104.761,172.242,38.313,157.260
C01166=1049.556,278.003,-104.730,172.239,38.310,157.259
C01167=1049.549,277.755,-104.699,172.236,38.307,157.258
C01168=1049.543,277.507,-104.669,172.234,38.303,157.257
C01169=1049.536,277.259,-104.637,172.230,38.301,157.257
C01170=1049.529,276.998,-104.605,172.227,38.297,157.256
C01171=1049.522,276.737,-104.572,172.224,38.294,157.255
C01172=1049.515,276.476,-104.540,172.221,38.291,157.254
C01173=1049.508,276.216,-104.508,172.217,38.287,157.254
C01174=1049.502,275.967,-104.477,172.215,38.285,157.253
C01175=1049.495,275.719,-104.447,172.212,38.281,157.252
C01176=1049.489,275.471,-104.416,172.209,38.278,157.251
C01177=1049.483,275.223,-104.385,172.206,38.275,157.251
C01178=1049.476,274.975,-104.355,172.203,38.272,157.250
C01179=1049.470,274.727,-104.324,172.200,38.269,157.249
C01180=1049.463,274.479,-104.293,172.197,38.266,157.249
C01181=1049.456,274.231,-104.263,172.195,38.263,157.248
C01182=1049.450,273.983,-104.232,172.191,38.260,157.247
C01183=1049.444,273.734,-104.202,172.188,38.257,157.246
C01184=1049.437,273.487,-104.172,172.186,38.254,157.246
C01185=1049.430,273.239,-104.141,172.182,38.251,157.245
C01186=1049.424,272.990,-104.110,172.180,38.248,157.244
C01187=1049.417,272.743,-104.080,172.177,38.244,157.244
C01188=1049.411,272.494,-104.049,172.173,38.242,157.243
C01189=1049.405,272.247,-104.019,172.171,38.239,157.242
C01190=1049.398,271.998,-103.989,172.168,38.235,157.241
C01191=1049.392,271.750,-103.958,172.165,38.232,157.241
C01192=1049.385,271.502,-103.928,172.162,38.229,157.240
C01193=1049.379,271.254,-103.898,172.159,38.227,157.239
C01194=1049.372,271.006,-103.868,172.157,38.223,157.239
C01195=1049.366,270.758,-103.837,172.153,38.220,157.238
C01196=1049.358,270.510,-103.807,172.151,38.217,157.237
C01197=1049.353,270.262,-103.777,172.148,38.214,157.236
C01198=1049.345,270.013,-103.747,172.144,38.211,157.236
C01199=1049.340,269.766,-103.716,172.142,38.208,157.235
C01200=1049.333,269.517,-103.686,172.139,38.205,157.234
C01201=1049.327,269.270,-103.656,172.137,38.202,157.234
C01202=1049.320,269.021,-103.626,172.133,38.199,157.233
C01203=1049.314,268.774,-103.595,172.131,38.196,157.232
C01204=1049.307,268.525,-103.565,172.128,38.193,157.232
C01205=1049.301,268.278,-103.535,172.124,38.190,157.231
C01206=1049.294,268.029,-103.505,172.122,38.187,157.230
C01207=1049.288,267.782,-103.474,172.119,38.184,157.229
C01208=1049.281,267.533,-103.445,172.117,38.181,157.229
C01209=1049.275,267.285,-103.415,172.113,38.178,157.228
C01210=1049.268,267.037,-103.384,172.110,38.175,157.227
C01211=1049.261,266.789,-103.355,172.108,38.172,157.227
C01212=1049.255,266.541,-103.324,172.105,38.169,157.226
C01213=1049.249,266.293,-103.295,172.102,38.166,157.225
C01214=1049.242,266.044,-103.265,172.099,38.163,157.224
C01215=1049.236,265.796,-103.235,172.097,38.160,157.224
C01216=1049.229,265.548,-103.205,172.094,38.157,157.223
C01217=1049.222,265.300,-103.175,172.091,38.154,157.222
C01218=1049.216,265.052,-103.145,172.088,38.151,157.222
C01219=1049.209,264.804,-103.115,172.085,38.148,157.221
C01220=1049.203,264.555,-103.085,172.083,38.145,157.220
C01221=1049.197,264.307,-103.055,172.080,38.142,157.220
C01222=1049.190,264.060,-103.025,172.077,38.139,157.219
C01223=1049.183,263.811,-102.996,172.074,38.136,157.218
C01224=1049.177,263.563,-102.966,172.071,38.133,157.217
C01225=1049.171,263.314,-102.936,172.069,38.130,157.217
C01226=1049.164,263.058,-102.906,172.066,38.127,157.216
C01227=1049.157,262.801,-102.875,172.063,38.124,157.215
C01228=1049.150,262.544,-102.844,172.060,38.121,157.215
C01229=1049.143,262.288,-102.813,172.058,38.118,157.214
C01230=1049.137,262.040,-102.784,172.055,38.115,157.213
C01231=1049.130,261.791,-102.754,172.051,38.112,157.213
C01232=1049.123,261.544,-102.725,172.049,38.108,157.212
C01233=1049.117,261.295,-102.695,172.046,38.106,157.211
C01234=1049.110,261.048,-102.665,172.044,38.103,157.210
C01235=1049.104,260.800,-102.636,172.041,38.100,157.210
C01236=1049.097,260.551,-102.607,172.038,38.097,157.209
C01237=1049.090,260.303,-102.577,172.035,38.094,157.208
C01238=1049.084,260.054,-102.548,172.033,38.091,157.208
C01239=1049.077,259.806,-102.519,172.030,38.088,157.207
C01240=1049.071,259.559,-102.489,172.027,38.085,157.206
C01241=1049.064,259.310,-102.460,172.024,38.082,157.206
C01242=1049.058,259.062,-102.431,172.021,38.080,157.205
C01243=1049.050,258.814,-102.400,172.019,38.077,157.204
C01244=1049.044,258.565,-102.371,172.016,38.074,157.204
C01245=1049.038,258.317,-102.342,172.014,38.071,157.203
C01246=1049.031,258.069,-102.312,172.011,38.068,157.202
C01247=1049.025,257.821,-102.283,172.009,38.065,157.202
C01248=1049.018,257.573,-102.254,172.005,38.062,157.201
C01249=1049.011,257.324,-102.225,172.002,38.059,157.200
C01250=1049.005,257.076,-102.195,172.000,38.056,157.200
C01251=1048.999,256.828,-102.166,171.997,38.053,157.199
C01252=1048.992,256.579,-102.137,171.995,38.050,157.198
C01253=1048.986,256.331,-102.107,171.992,38.047,157.198
C01254=1048.979,256.084,-102.079,171.990,38.044,157.197
C01255=1048.971,255.835,-102.049,171.987,38.041,157.196
C01256=1048.965,255.587,-102.020,171.984,38.038,157.196
C01257=1048.959,255.339,-101.991,171.981,38.036,157.195
C01258=1048.953,255.091,-101.962,171.979,38.033,157.194
C01259=1048.946,254.842,-101.932,171.976,38.030,157.194
C01260=1048.940,254.594,-101.903,171.973,38.026,157.193
C01261=1048.933,254.346,-101.874,171.971,38.023,157.192
C01262=1048.927,254.098,-101.845,171.968,38.020,157.192
C01263=1048.920,253.849,-101.816,171.966,38.018,157.191
C01264=1048.914,253.601,-101.787,171.963,38.015,157.190
C01265=1048.907,253.353,-101.757,171.961,38.012,157.190
C01266=1048.901,253.105,-101.728,171.958,38.009,157.189
C01267=1048.894,252.857,-101.700,171.955,38.006,157.188
C01268=1048.887,252.608,-101.670,171.952,38.003,157.188
C01269=1048.881,252.360,-101.641,171.950,38.000,157.187
C01270=1048.875,252.112,-101.612,171.947,37.997,157.186
C01271=1048.869,251.864,-101.583,171.944,37.994,157.185
C01272=1048.862,251.616,-101.554,171.942,37.991,157.185
C01273=1048.856,251.366,-101.525,171.939,37.988,157.184
C01274=1048.850,251.118,-101.496,171.937,37.985,157.183
C01275=1048.843,250.870,-101.467,171.934,37.982,157.183
C01276=1048.836,250.622,-101.439,171.932,37.979,157.182
C01277=1048.830,250.374,-101.410,171.929,37.976,157.181
C01278=1048.824,250.126,-101.381,171.927,37.973,157.181
C01279=1048.818,249.878,-101.352,171.924,37.970,157.180
C01280=1048.811,249.630,-101.323,171.922,37.967,157.179
C01281=1048.804,249.381,-101.293,171.919,37.964,157.179
C01282=1048.798,249.123,-101.264,171.917,37.961,157.178
C01283=1048.792,248.865,-101.233,171.914,37.958,157.177
C01284=1048.785,248.606,-101.203,171.911,37.955,157.177
C01285=1048.778,248.348,-101.174,171.909,37.952,157.176
C01286=1048.772,248.099,-101.145,171.906,37.948,157.175
C01287=1048.766,247.851,-101.116,171.904,37.945,157.174
C01288=1048.760,247.603,-101.087,171.901,37.942,157.174
C01289=1048.753,247.355,-101.058,171.899,37.939,157.173
C01290=1048.747,247.107,-101.030,171.896,37.937,157.172
C01291=1048.740,246.858,-101.001,171.894,37.934,157.172
C01292=1048.734,246.610,-100.972,171.891,37.930,157.171
C01293=1048.728,246.362,-100.943,171.888,37.927,157.170
C01294=1048.722,246.113,-100.914,171.886,37.924,157.170
C01295=1048.716,245.865,-100.885,171.883,37.921,157.169
C01296=1048.709,245.617,-100.857,171.881,37.918,157.168
C01297=1048.703,245.369,-100.829,171.878,37.915,157.168
C01298=1048.696,245.121,-100.800,171.876,37.913,157.167
C01299=1048.689,244.872,-100.771,171.873,37.910,157.166
C01300=1048.683,244.623,-100.742,171.871,37.907,157.166
C01301=1048.676,244.376,-100.714,171.868,37.903,157.165
C01302=1048.670,244.127,-100.686,171.866,37.900,157.164
C01303=1048.664,243.879,-100.657,171.863,37.897,157.164
C01304=1048.657,243.630,-100.629,171.861,37.894,157.163
C01305=1048.651,243.382,-100.600,171.858,37.892,157.162
C01306=1048.644,243.134,-100.572,171.856,37.889,157.162
C01307=1048.638,242.885,-100.543,171.853,37.886,157.161
C01308=1048.632,242.637,-100.515,171.851,37.883,157.160
C01309=1048.625,242.389,-100.486,171.848,37.880,157.160
C01310=1048.619,242.140,-100.458,171.845,37.877,157.159
C01311=1048.612,241.892,-100.430,171.844,37.874,157.158
C01312=1048.606,241.644,-100.401,171.841,37.870,157.158
C01313=1048.599,241.396,-100.373,171.839,37.867,157.157
C01314=1048.593,241.147,-100.345,171.836,37.865,157.156
C01315=1048.587,240.899,-100.317,171.834,37.862,157.156
C01316=1048.580,240.650,-100.288,171.831,37.859,157.155
C01317=1048.574,240.402,-100.260,171.829,37.856,157.154
C01318=1048.567,240.154,-100.232,171.826,37.853,157.154
C01319=1048.561,239.905,-100.203,171.824,37.850,157.153
C01320=1048.554,239.657,-100.176,171.821,37.847,157.152
C01321=1048.547,239.409,-100.147,171.819,37.844,157.152
C01322=1048.541,239.160,-100.119,171.816,37.841,157.151
C01323=1048.534,238.912,-100.091,171.814,37.838,157.150
C01324=1048.528,238.664,-100.063,171.812,37.835,157.150
C01325=1048.522,238.416,-100.035,171.810,37.832,157.149
C01326=1048.515,238.168,-100.007,171.807,37.829,157.148
C01327=1048.509,237.919,-99.979,171.805,37.826,157.148
C01328=1048.503,237.670,-99.951,171.802,37.824,157.147
C01329=1048.496,237.423,-99.922,171.800,37.821,157.146
C01330=1048.489,237.174,-99.895,171.797,37.818,157.146
C01331=1048.483,236.925,-99.866,171.795,37.815,157.145
C01332=1048.476,236.677,-99.839,171.792,37.812,157.144
C01333=1048.470,236.429,-99.811,171.791,37.809,157.144
C01334=1048.463,236.180,-99.783,171.788,37.806,157.143
C01335=1048.457,235.932,-99.754,171.786,37.803,157.142
C01336=1048.450,235.684,-99.726,171.783,37.800,157.142
C01337=1048.443,235.435,-99.699,171.781,37.797,157.141
C01338=1048.437,235.171,-99.670,171.778,37.794,157.140
C01339=1048.430,234.907,-99.640,171.775,37.791,157.140
C01340=1048.423,234.643,-99.610,171.773,37.788,157.139
C01341=1048.417,234.379,-99.581,171.770,37.784,157.138
C01342=1048.411,234.130,-99.552,171.768,37.781,157.138
C01343=1048.404,233.882,-99.524,171.766,37.778,157.137
C01344=1048.397,233.633,-99.497,171.764,37.775,157.136
C01345=1048.391,233.385,-99.469,171.761,37.772,157.136
C01346=1048.385,233.136,-99.441,171.759,37.769,157.135
C01347=1048.379,232.888,-99.413,171.756,37.766,157.134
C01348=1048.372,232.640,-99.386,171.754,37.764,157.134
C01349=1048.365,232.392,-99.358,171.752,37.761,157.133
C01350=1048.359,232.143,-99.330,171.750,37.758,157.132
C01351=1048.353,231.894,-99.302,171.747,37.755,157.132
C01352=1048.346,231.646,-99.274,171.745,37.752,157.131
C01353=1048.340,231.398,-99.247,171.742,37.749,157.130
C01354=1048.333,231.150,-99.219,171.740,37.746,157.130
C01355=1048.327,230.901,-99.191,171.738,37.743,157.129
C01356=1048.320,230.653,-99.164,171.736,37.740,157.128
C01357=1048.313,230.404,-99.136,171.733,37.737,157.128
C01358=1048.307,230.157,-99.108,171.731,37.733,157.127
C01359=1048.301,229.908,-99.081,171.728,37.731,157.126
C01360=1048.295,229.659,-99.053,171.727,37.728,157.126
C01361=1048.288,229.410,-99.025,171.724,37.725,157.125
C01362=1048.282,229.163,-98.998,171.722,37.722,157.124
C01363=1048.275,228.914,-98.970,171.719,37.719,157.124
C01364=1048.269,228.666,-98.943,171.718,37.716,157.123
C01365=1048.262,228.417,-98.916,171.715,37.713,157.122
C01366=1048.256,228.168,-98.888,171.713,37.710,157.122
C01367=1048.250,227.921,-98.860,171.710,37.707,157.121
C01368=1048.243,227.672,-98.834,171.708,37.704,157.121
C01369=1048.236,227.423,-98.806,171.706,37.701,157.120
C01370=1048.229,227.175,-98.779,171.704,37.698,157.119
C01371=1048.223,226.927,-98.751,171.701,37.695,157.119
C01372=1048.217,226.678,-98.724,171.699,37.692,157.118
C01373=1048.210,226.430,-98.696,171.697,37.689,157.117
C01374=1048.203,226.181,-98.669,171.695,37.686,157.117
C01375=1048.198,225.933,-98.642,171.692,37.683,157.116
C01376=1048.191,225.684,-98.614,171.690,37.680,157.115
C01377=1048.184,225.436,-98.588,171.688,37.677,157.115
C01378=1048.177,225.187,-98.560,171.686,37.674,157.114
C01379=1048.171,224.939,-98.533,171.683,37.671,157.113
C01380=1048.165,224.690,-98.506,171.681,37.669,157.113
C01381=1048.158,224.442,-98.478,171.679,37.666,157.112
C01382=1048.152,224.194,-98.451,171.677,37.663,157.111
C01383=1048.145,223.945,-98.424,171.674,37.660,157.111
C01384=1048.139,223.697,-98.396,171.672,37.657,157.110
C01385=1048.132,223.449,-98.370,171.670,37.654,157.110
C01386=1048.126,223.200,-98.342,171.668,37.651,157.109
C01387=1048.119,222.951,-98.315,171.665,37.648,157.108
C01388=1048.113,222.703,-98.288,171.663,37.644,157.107
C01389=1048.107,222.454,-98.261,171.661,37.641,157.107
C01390=1048.100,222.206,-98.233,171.659,37.638,157.106
C01391=1048.094,221.958,-98.207,171.656,37.635,157.106
C01392=1048.087,221.709,-98.179,171.655,37.632,157.105
C01393=1048.081,221.461,-98.153,171.652,37.629,157.104
C01394=1048.074,221.189,-98.123,171.650,37.626,157.103
C01395=1048.067,220.918,-98.093,171.647,37.623,157.103
C01396=1048.060,220.646,-98.063,171.645,37.619,157.102
C01397=1048.053,220.374,-98.034,171.643,37.616,157.101
C01398=1048.046,220.125,-98.007,171.641,37.613,157.101
C01399=1048.040,219.877,-97.981,171.638,37.610,157.100
C01400=1048.033,219.629,-97.953,171.637,37.607,157.099
C01401=1048.026,219.380,-97.926,171.634,37.605,157.099
C01402=1048.020,219.132,-97.900,171.632,37.602,157.098
C01403=1048.014,218.883,-97.872,171.629,37.599,157.097
C01404=1048.007,218.635,-97.846,171.628,37.596,157.097
C01405=1048.001,218.386,-97.819,171.625,37.593,157.096
C01406=1047.994,218.137,-97.793,171.623,37.590,157.096
C01407=1047.988,217.890,-97.765,171.621,37.587,157.095
C01408=1047.981,217.641,-97.738,171.619,37.583,157.094
C01409=1047.975,217.393,-97.712,171.616,37.580,157.093
C01410=1047.968,217.144,-97.685,171.615,37.577,157.093
C01411=1047.961,216.895,-97.658,171.612,37.574,157.092
C01412=1047.955,216.647,-97.631,171.610,37.571,157.092
C01413=1047.948,216.398,-97.605,171.608,37.568,157.091
C01414=1047.942,216.150,-97.578,171.606,37.565,157.090
C01415=1047.936,215.901,-97.551,171.604,37.562,157.090
C01416=1047.929,215.653,-97.524,171.602,37.559,157.089
C01417=1047.923,215.404,-97.497,171.599,37.556,157.088
C01418=1047.916,215.156,-97.471,171.598,37.553,157.088
C01419=1047.910,214.907,-97.444,171.595,37.550,157.087
C01420=1047.903,214.659,-97.418,171.593,37.547,157.086
C01421=1047.897,214.410,-97.391,171.591,37.544,157.086
C01422=1047.891,214.162,-97.365,171.589,37.541,157.085
C01423=1047.884,213.914,-97.337,171.587,37.538,157.084
C01424=1047.878,213.665,-97.311,171.585,37.535,157.084
C01425=1047.871,213.417,-97.284,171.582,37.532,157.083
C01426=1047.865,213.168,-97.258,171.581,37.529,157.082
C01427=1047.858,212.919,-97.231,171.578,37.526,157.082
C01428=1047.852,212.671,-97.205,171.577,37.523,157.081
C01429=1047.845,212.422,-97.178,171.574,37.519,157.080
C01430=1047.839,212.174,-97.152,171.572,37.517,157.080
C01431=1047.832,211.925,-97.125,171.570,37.514,157.079
C01432=1047.826,211.677,-97.099,171.568,37.511,157.078
C01433=1047.819,211.428,-97.072,171.566,37.508,157.078
C01434=1047.814,211.180,-97.045,171.564,37.505,157.077
C01435=1047.806,210.931,-97.019,171.562,37.502,157.077
C01436=1047.800,210.683,-96.993,171.560,37.499,157.076
C01437=1047.794,210.434,-96.966,171.558,37.496,157.075
C01438=1047.787,210.186,-96.940,171.556,37.492,157.074
C01439=1047.781,209.938,-96.913,171.554,37.489,157.074
C01440=1047.774,209.689,-96.887,171.552,37.486,157.073
C01441=1047.768,209.440,-96.862,171.550,37.483,157.073
C01442=1047.762,209.191,-96.835,171.547,37.480,157.072
C01443=1047.755,208.943,-96.808,171.546,37.477,157.071
C01444=1047.748,208.694,-96.782,171.543,37.474,157.071
C01445=1047.741,208.446,-96.756,171.542,37.471,157.070
C01446=1047.736,208.198,-96.729,171.539,37.468,157.069
C01447=1047.729,207.949,-96.703,171.538,37.465,157.069
C01448=1047.722,207.700,-96.678,171.535,37.462,157.068
C01449=1047.716,207.451,-96.651,171.534,37.459,157.067
C01450=1047.709,207.185,-96.623,171.531,37.456,157.067
C01451=1047.702,206.919,-96.594,171.529,37.452,157.066
C01452=1047.695,206.654,-96.567,171.527,37.449,157.065
C01453=1047.688,206.387,-96.539,171.525,37.446,157.064
C01454=1047.662,205.335,-96.432,171.280,37.347,157.042
C01455=1047.656,205.087,-96.407,171.278,37.344,157.041
C01456=1047.650,204.838,-96.383,171.275,37.343,157.041
C01457=1047.644,204.589,-96.357,171.272,37.340,157.040
C01458=1047.638,204.340,-96.332,171.270,37.338,157.040
C01459=1047.631,204.092,-96.307,171.267,37.336,157.039
C01460=1047.625,203.843,-96.283,171.264,37.333,157.039
C01461=1047.619,203.595,-96.258,171.262,37.331,157.038
C01462=1047.613,203.346,-96.232,171.259,37.329,157.038
C01463=1047.607,203.097,-96.207,171.256,37.327,157.037
C01464=1047.601,202.848,-96.182,171.254,37.324,157.037
C01465=1047.595,202.600,-96.157,171.252,37.322,157.036
C01466=1047.589,202.351,-96.132,171.248,37.320,157.036
C01467=1047.583,202.102,-96.107,171.246,37.318,157.036
C01468=1047.577,201.854,-96.082,171.244,37.315,157.035
C01469=1047.571,201.606,-96.057,171.240,37.313,157.034
C01470=1047.566,201.356,-96.032,171.238,37.311,157.034
C01471=1047.559,201.108,-96.008,171.236,37.309,157.034
C01472=1047.553,200.859,-95.983,171.232,37.306,157.033
C01473=1047.546,200.610,-95.958,171.230,37.305,157.033
C01474=1047.540,200.362,-95.934,171.228,37.302,157.032
C01475=1047.534,200.113,-95.909,171.224,37.300,157.032
C01476=1047.528,199.864,-95.885,171.222,37.298,157.031
C01477=1047.521,199.615,-95.859,171.220,37.296,157.031
C01478=1047.515,199.366,-95.835,171.217,37.294,157.030
C01479=1047.509,199.118,-95.810,171.214,37.291,157.030
C01480=1047.503,198.869,-95.786,171.212,37.290,157.030
C01481=1047.496,198.621,-95.761,171.209,37.287,157.029
C01482=1047.490,198.371,-95.736,171.206,37.286,157.029
C01483=1047.484,198.123,-95.713,171.204,37.283,157.028
C01484=1047.478,197.875,-95.687,171.201,37.281,157.028
C01485=1047.472,197.626,-95.663,171.199,37.279,157.027
C01486=1047.466,197.378,-95.638,171.196,37.277,157.027
C01487=1047.460,197.128,-95.614,171.193,37.275,157.026
C01488=1047.453,196.879,-95.590,171.191,37.272,157.026
C01489=1047.447,196.631,-95.564,171.188,37.271,157.025
C01490=1047.441,196.382,-95.541,171.185,37.268,157.025
C01491=1047.435,196.133,-95.516,171.183,37.266,157.025
C01492=1047.428,195.885,-95.491,171.181,37.264,157.024
C01493=1047.423,195.636,-95.467,171.178,37.262,157.024
C01494=1047.417,195.387,-95.442,171.175,37.260,157.023
C01495=1047.410,195.139,-95.418,171.173,37.258,157.023
C01496=1047.405,194.890,-95.393,171.171,37.256,157.022
C01497=1047.398,194.641,-95.369,171.167,37.254,157.022
C01498=1047.393,194.392,-95.345,171.165,37.251,157.021
C01499=1047.386,194.144,-95.320,171.163,37.250,157.021
C01500=1047.380,193.895,-95.296,171.160,37.247,157.020
C01501=1047.374,193.646,-95.272,171.158,37.245,157.020
C01502=1047.368,193.397,-95.247,171.155,37.243,157.020
C01503=1047.362,193.148,-95.222,171.152,37.241,157.019
C01504=1047.356,192.900,-95.198,171.150,37.239,157.019
C01505=1047.350,192.651,-95.174,171.148,37.237,157.018
C01506=1047.344,192.403,-95.150,171.144,37.235,157.018
C01507=1047.338,192.153,-95.126,171.142,37.233,157.017
C01508=1047.332,191.905,-95.102,171.140,37.231,157.017
C01509=1047.326,191.656,-95.077,171.138,37.229,157.017
C01510=1047.319,191.407,-95.053,171.135,37.226,157.016
C01511=1047.314,191.159,-95.028,171.132,37.225,157.016
C01512=1047.307,190.910,-95.004,171.130,37.222,157.015
C01513=1047.302,190.661,-94.980,171.127,37.220,157.015
C01514=1047.295,190.412,-94.956,171.125,37.219,157.014
C01515=1047.289,190.129,-94.928,171.122,37.216,157.014
C01516=1047.282,189.844,-94.900,171.119,37.214,157.013
C01517=1047.275,189.559,-94.873,171.116,37.211,157.013
C01518=1047.268,189.275,-94.845,171.114,37.209,157.012
C01519=1047.263,189.026,-94.821,171.111,37.207,157.012
C01520=1047.256,188.778,-94.797,171.108,37.205,157.011
C01521=1047.251,188.528,-94.772,171.106,37.202,157.011
C01522=1047.245,188.280,-94.749,171.103,37.201,157.011
C01523=1047.239,188.031,-94.724,171.101,37.198,157.010
C01524=1047.233,187.783,-94.700,171.099,37.196,157.010
C01525=1047.227,187.533,-94.676,171.096,37.195,157.009
C01526=1047.221,187.285,-94.652,171.094,37.192,157.009
C01527=1047.215,187.036,-94.628,171.091,37.190,157.008
C01528=1047.209,186.787,-94.604,171.089,37.188,157.008
C01529=1047.203,186.539,-94.580,171.086,37.186,157.008
C01530=1047.197,186.290,-94.556,171.084,37.184,157.007
C01531=1047.191,186.041,-94.533,171.082,37.182,157.007
C01532=1047.185,185.792,-94.508,171.079,37.180,157.006
C01533=1047.179,185.543,-94.484,171.077,37.178,157.006
C01534=1047.173,185.294,-94.460,171.074,37.176,157.005
C01535=1047.167,185.046,-94.436,171.071,37.174,157.005
C01536=1047.162,184.797,-94.412,171.069,37.172,157.005
C01537=1047.155,184.548,-94.388,171.067,37.170,157.004
C01538=1047.150,184.300,-94.364,171.065,37.168,157.004
C01539=1047.144,184.051,-94.341,171.062,37.166,157.003
C01540=1047.138,183.802,-94.317,171.060,37.163,157.003
C01541=1047.132,183.554,-94.293,171.058,37.162,157.002
C01542=1047.125,183.304,-94.270,171.054,37.160,157.002
C01543=1047.119,183.056,-94.246,171.052,37.158,157.002
C01544=1047.113,182.807,-94.222,171.050,37.156,157.001
C01545=1047.107,182.558,-94.199,171.048,37.154,157.001
C01546=1047.100,182.309,-94.175,171.045,37.153,157.000
C01547=1047.094,182.061,-94.151,171.043,37.151,157.000
C01548=1047.088,181.811,-94.128,171.040,37.149,157.000
C01549=1047.082,181.563,-94.104,171.037,37.147,156.999
C01550=1047.075,181.314,-94.080,171.035,37.145,156.999
C01551=1047.069,181.065,-94.057,171.033,37.143,156.998
C01552=1047.063,180.816,-94.033,171.031,37.141,156.998
C01553=1047.057,180.567,-94.010,171.028,37.139,156.998
C01554=1047.051,180.319,-93.987,171.026,37.137,156.997
C01555=1047.045,180.069,-93.963,171.023,37.136,156.997
C01556=1047.038,179.821,-93.940,171.021,37.134,156.997
C01557=1047.031,179.572,-93.916,171.018,37.132,156.996
C01558=1047.026,179.323,-93.893,171.016,37.130,156.996
C01559=1047.019,179.075,-93.870,171.014,37.128,156.995
C01560=1047.013,178.825,-93.846,171.012,37.126,156.995
C01561=1047.007,178.577,-93.823,171.009,37.124,156.995
C01562=1047.001,178.327,-93.799,171.007,37.122,156.994
C01563=1046.995,178.079,-93.776,171.004,37.121,156.994
C01564=1046.989,177.830,-93.753,171.002,37.119,156.993
C01565=1046.982,177.581,-93.729,170.999,37.117,156.993
C01566=1046.977,177.332,-93.706,170.997,37.115,156.993
C01567=1046.970,177.084,-93.683,170.995,37.113,156.992
C01568=1046.964,176.835,-93.659,170.992,37.112,156.992
C01569=1046.958,176.586,-93.636,170.990,37.110,156.992
C01570=1046.952,176.338,-93.613,170.988,37.108,156.991
C01571=1046.945,176.088,-93.589,170.986,37.106,156.991
C01572=1046.940,175.839,-93.567,170.983,37.104,156.990
C01573=1046.934,175.591,-93.543,170.981,37.102,156.990
C01574=1046.927,175.341,-93.520,170.978,37.100,156.990
C01575=1046.921,175.093,-93.496,170.976,37.098,156.989
C01576=1046.915,174.844,-93.474,170.973,37.097,156.989
C01577=1046.909,174.595,-93.451,170.971,37.095,156.988
C01578=1046.902,174.347,-93.427,170.969,37.093,156.988
C01579=1046.896,174.062,-93.400,170.967,37.091,156.988
C01580=1046.889,173.777,-93.374,170.963,37.089,156.987
C01581=1046.882,173.492,-93.347,170.961,37.087,156.987
C01582=1046.875,173.207,-93.321,170.959,37.084,156.986
C01583=1046.869,172.958,-93.298,170.956,37.083,156.986
C01584=1046.863,172.709,-93.274,170.954,37.081,156.986
C01585=1046.857,172.461,-93.251,170.952,37.079,156.985
C01586=1046.851,172.212,-93.228,170.950,37.077,156.985
C01587=1046.845,171.963,-93.205,170.947,37.075,156.984
C01588=1046.839,171.714,-93.182,170.944,37.074,156.984
C01589=1046.833,171.465,-93.158,170.942,37.072,156.984
C01590=1046.826,171.216,-93.136,170.940,37.070,156.983
C01591=1046.821,170.967,-93.113,170.937,37.068,156.983
C01592=1046.815,170.719,-93.089,170.935,37.066,156.983
C01593=1046.809,170.470,-93.067,170.933,37.065,156.982
C01594=1046.803,170.221,-93.043,170.931,37.063,156.982
C01595=1046.797,169.972,-93.020,170.928,37.061,156.981
C01596=1046.790,169.723,-92.998,170.926,37.059,156.981
C01597=1046.785,169.474,-92.975,170.924,37.057,156.981
C01598=1046.779,169.225,-92.952,170.921,37.055,156.980
C01599=1046.773,168.977,-92.928,170.919,37.053,156.980
C01600=1046.767,168.727,-92.905,170.917,37.051,156.979
C01601=1046.761,168.479,-92.882,170.915,37.049,156.979
C01602=1046.754,168.230,-92.860,170.912,37.048,156.979
C01603=1046.749,167.981,-92.837,170.910,37.046,156.978
C01604=1046.743,167.732,-92.814,170.908,37.044,156.978
C01605=1046.737,167.483,-92.791,170.906,37.042,156.978
C01606=1046.732,167.234,-92.768,170.903,37.040,156.977
C01607=1046.725,166.986,-92.746,170.901,37.039,156.977
C01608=1046.719,166.737,-92.723,170.899,37.037,156.976
C01609=1046.713,166.487,-92.699,170.897,37.035,156.976
C01610=1046.707,166.238,-92.676,170.894,37.033,156.976
C01611=1046.702,165.989,-92.653,170.892,37.031,156.975
C01612=1046.696,165.741,-92.631,170.890,37.029,156.975
C01613=1046.689,165.492,-92.608,170.888,37.028,156.975
C01614=1046.684,165.243,-92.585,170.885,37.026,156.974
C01615=1046.678,164.994,-92.562,170.883,37.024,156.974
C01616=1046.672,164.745,-92.539,170.882,37.022,156.973
C01617=1046.666,164.496,-92.516,170.880,37.020,156.973
C01618=1046.660,164.248,-92.494,170.877,37.019,156.973
C01619=1046.654,163.999,-92.471,170.875,37.017,156.972
C01620=1046.648,163.750,-92.448,170.873,37.015,156.972
C01621=1046.643,163.501,-92.425,170.871,37.013,156.972
C01622=1046.636,163.253,-92.403,170.868,37.011,156.971
C01623=1046.631,163.004,-92.380,170.866,37.009,156.971
C01624=1046.625,162.755,-92.357,170.864,37.008,156.970
C01625=1046.619,162.506,-92.334,170.862,37.006,156.970
C01626=1046.613,162.257,-92.311,170.859,37.004,156.970
C01627=1046.607,162.008,-92.289,170.857,37.002,156.969
C01628=1046.601,161.759,-92.266,170.855,37.000,156.969
C01629=1046.596,161.510,-92.244,170.853,36.999,156.969
C01630=1046.590,161.261,-92.221,170.850,36.997,156.968
C01631=1046.584,161.012,-92.198,170.848,36.995,156.968
C01632=1046.578,160.764,-92.175,170.846,36.992,156.967
C01633=1046.572,160.514,-92.153,170.844,36.991,156.967
C01634=1046.566,160.265,-92.131,170.842,36.989,156.967
C01635=1046.560,160.017,-92.108,170.840,36.988,156.966
C01636=1046.554,159.767,-92.086,170.838,36.986,156.966
C01637=1046.548,159.518,-92.063,170.836,36.984,156.966
C01638=1046.542,159.270,-92.041,170.833,36.982,156.965
C01639=1046.535,159.021,-92.018,170.831,36.981,156.965
C01640=1046.530,158.772,-91.996,170.829,36.979,156.965
C01641=1046.523,158.523,-91.974,170.827,36.977,156.964
C01642=1046.518,158.274,-91.951,170.825,36.975,156.964
C01643=1046.511,157.989,-91.926,170.822,36.974,156.963
C01644=1046.504,157.703,-91.901,170.819,36.972,156.963
C01645=1046.496,157.418,-91.875,170.817,36.970,156.963
C01646=1046.489,157.133,-91.849,170.814,36.968,156.962
C01647=1046.484,156.884,-91.826,170.812,36.966,156.962
C01648=1046.477,156.634,-91.805,170.810,36.965,156.962
C01649=1046.471,156.386,-91.782,170.808,36.963,156.961
C01650=1046.465,156.137,-91.759,170.806,36.961,156.961
C01651=1046.460,155.888,-91.738,170.803,36.959,156.960
C01652=1046.453,155.640,-91.716,170.801,36.957,156.960
C01653=1046.448,155.390,-91.694,170.800,36.956,156.960
C01654=1046.441,155.142,-91.671,170.798,36.954,156.959
C01655=1046.435,154.893,-91.650,170.795,36.952,156.959
C01656=1046.429,154.644,-91.627,170.793,36.951,156.959
C01657=1046.423,154.394,-91.605,170.791,36.949,156.958
C01658=1046.417,154.146,-91.583,170.789,36.947,156.958
C01659=1046.411,153.897,-91.561,170.787,36.946,156.958
C01660=1046.405,153.648,-91.538,170.784,36.944,156.957
C01661=1046.399,153.399,-91.516,170.782,36.943,156.957
C01662=1046.392,153.150,-91.494,170.780,36.941,156.957
C01663=1046.386,152.901,-91.472,170.778,36.939,156.956
C01664=1046.381,152.651,-91.450,170.775,36.937,156.956
C01665=1046.374,152.403,-91.428,170.774,36.936,156.956
C01666=1046.369,152.154,-91.407,170.772,36.934,156.955
C01667=1046.362,151.906,-91.384,170.770,36.932,156.955
C01668=1046.357,151.656,-91.362,170.767,36.930,156.955
C01669=1046.351,151.407,-91.340,170.765,36.929,156.954
C01670=1046.344,151.158,-91.318,170.763,36.927,156.954
C01671=1046.338,150.909,-91.296,170.761,36.926,156.954
C01672=1046.331,150.660,-91.274,170.759,36.924,156.953
C01673=1046.326,150.411,-91.252,170.756,36.923,156.953
C01674=1046.320,150.162,-91.231,170.755,36.921,156.953
C01675=1046.314,149.914,-91.208,170.753,36.919,156.952
C01676=1046.308,149.665,-91.187,170.751,36.918,156.952
C01677=1046.302,149.415,-91.165,170.749,36.916,156.952
C01678=1046.295,149.166,-91.143,170.746,36.914,156.951
C01679=1046.290,148.917,-91.120,170.744,36.912,156.951
C01680=1046.284,148.668,-91.099,170.742,36.911,156.951
C01681=1046.278,148.420,-91.077,170.740,36.909,156.950
C01682=1046.272,148.170,-91.056,170.737,36.907,156.950
C01683=1046.265,147.922,-91.033,170.736,36.906,156.950
C01684=1046.259,147.673,-91.012,170.734,36.904,156.949
C01685=1046.253,147.423,-90.990,170.732,36.902,156.949
C01686=1046.247,147.174,-90.969,170.729,36.901,156.949
C01687=1046.241,146.926,-90.947,170.727,36.899,156.948
C01688=1046.235,146.677,-90.925,170.725,36.898,156.948
C01689=1046.229,146.428,-90.903,170.723,36.896,156.948
C01690=1046.223,146.179,-90.882,170.721,36.894,156.947
C01691=1046.216,145.929,-90.860,170.719,36.893,156.947
C01692=1046.210,145.680,-90.838,170.717,36.891,156.947
C01693=1046.205,145.432,-90.817,170.715,36.890,156.946
C01694=1046.198,145.183,-90.795,170.713,36.888,156.946
C01695=1046.192,144.934,-90.773,170.711,36.887,156.946
C01696=1046.186,144.685,-90.751,170.708,36.885,156.945
C01697=1046.180,144.436,-90.730,170.706,36.883,156.945
C01698=1046.174,144.187,-90.709,170.705,36.882,156.945
C01699=1046.168,143.938,-90.687,170.703,36.880,156.944
C01700=1046.162,143.689,-90.665,170.701,36.879,156.944
C01701=1046.156,143.439,-90.644,170.698,36.877,156.944
C01702=1046.150,143.190,-90.622,170.696,36.875,156.943
C01703=1046.144,142.942,-90.601,170.694,36.874,156.943
C01704=1046.138,142.693,-90.579,170.692,36.872,156.943
C01705=1046.132,142.443,-90.557,170.691,36.871,156.943
C01706=1046.125,142.194,-90.536,170.688,36.869,156.942
C01707=1046.118,141.909,-90.511,170.686,36.867,156.942
C01708=1046.111,141.623,-90.487,170.684,36.865,156.941
C01709=1046.105,141.338,-90.462,170.681,36.863,156.941
C01710=1046.097,141.053,-90.438,170.678,36.861,156.941
C01711=1046.091,140.804,-90.416,170.676,36.860,156.940
C01712=1046.085,140.555,-90.394,170.675,36.858,156.940
C01713=1046.079,140.305,-90.373,170.673,36.857,156.940
C01714=1046.074,140.056,-90.352,170.670,36.855,156.939
C01715=1046.067,139.807,-90.330,170.668,36.854,156.939
C01716=1046.061,139.558,-90.309,170.666,36.852,156.939
C01717=1046.056,139.309,-90.288,170.665,36.850,156.938
C01718=1046.049,139.061,-90.267,170.663,36.849,156.938
C01719=1046.043,138.811,-90.245,170.660,36.847,156.938
C01720=1046.037,138.562,-90.223,170.658,36.846,156.937
C01721=1046.031,138.314,-90.202,170.656,36.844,156.937
C01722=1046.024,138.064,-90.182,170.654,36.842,156.937
C01723=1046.018,137.815,-90.160,170.653,36.841,156.937
C01724=1046.013,137.566,-90.139,170.650,36.839,156.936
C01725=1046.006,137.317,-90.117,170.648,36.838,156.936
C01726=1046.000,137.068,-90.095,170.646,36.836,156.936
C01727=1045.994,136.820,-90.075,170.644,36.835,156.935
C01728=1045.988,136.570,-90.054,170.642,36.833,156.935
C01729=1045.982,136.321,-90.032,170.640,36.831,156.935
C01730=1045.976,136.073,-90.012,170.638,36.830,156.934
C01731=1045.970,135.823,-89.990,170.636,36.828,156.934
C01732=1045.964,135.574,-89.969,170.634,36.827,156.934
C01733=1045.957,135.325,-89.948,170.632,36.825,156.933
C01734=1045.951,135.076,-89.927,170.630,36.823,156.933
C01735=1045.945,134.827,-89.905,170.628,36.822,156.933
C01736=1045.939,134.578,-89.885,170.626,36.820,156.932
C01737=1045.933,134.329,-89.863,170.624,36.819,156.932
C01738=1045.927,134.080,-89.842,170.622,36.817,156.932
C01739=1045.921,133.831,-89.822,170.620,36.816,156.932
C01740=1045.915,133.582,-89.800,170.618,36.814,156.931
C01741=1045.908,133.332,-89.779,170.616,36.812,156.931
C01742=1045.902,133.084,-89.759,170.614,36.811,156.931
C01743=1045.896,132.834,-89.737,170.612,36.809,156.930
C01744=1045.891,132.586,-89.716,170.610,36.808,156.930
C01745=1045.884,132.336,-89.695,170.608,36.806,156.930
C01746=1045.878,132.087,-89.674,170.606,36.805,156.929
C01747=1045.872,131.839,-89.653,170.604,36.803,156.929
C01748=1045.866,131.589,-89.632,170.602,36.802,156.929
C01749=1045.860,131.341,-89.611,170.600,36.800,156.928
C01750=1045.854,131.091,-89.590,170.598,36.799,156.928
C01751=1045.847,130.842,-89.569,170.596,36.797,156.928
C01752=1045.841,130.593,-89.549,170.594,36.796,156.928
C01753=1045.835,130.344,-89.527,170.592,36.795,156.927
C01754=1045.829,130.094,-89.507,170.591,36.793,156.927
C01755=1045.822,129.846,-89.486,170.588,36.792,156.927
C01756=1045.817,129.596,-89.465,170.586,36.790,156.926
C01757=1045.810,129.348,-89.445,170.584,36.788,156.926
C01758=1045.804,129.098,-89.424,170.582,36.787,156.926
C01759=1045.797,128.850,-89.403,170.581,36.785,156.925
C01760=1045.791,128.601,-89.383,170.578,36.784,156.925
C01761=1045.785,128.352,-89.361,170.576,36.782,156.925
C01762=1045.779,128.103,-89.341,170.574,36.781,156.925
C01763=1045.772,127.854,-89.320,170.572,36.780,156.924
C01764=1045.767,127.604,-89.299,170.571,36.778,156.924
C01765=1045.760,127.356,-89.279,170.568,36.777,156.924
C01766=1045.754,127.106,-89.258,170.566,36.775,156.923
C01767=1045.748,126.857,-89.238,170.564,36.774,156.923
C01768=1045.742,126.608,-89.217,170.562,36.773,156.923
C01769=1045.736,126.359,-89.196,170.561,36.771,156.923
C01770=1045.729,126.110,-89.175,170.559,36.769,156.922
C01771=1045.719,125.691,-89.141,170.555,36.767,156.922
C01772=1045.709,125.273,-89.107,170.552,36.765,156.921
C01773=1045.698,124.855,-89.072,170.549,36.762,156.921
C01774=1045.688,124.436,-89.037,170.545,36.759,156.920
C01775=1045.682,124.188,-89.016,170.543,36.758,156.920
C01776=1045.676,123.938,-88.996,170.541,36.757,156.920
C01777=1045.670,123.689,-88.976,170.540,36.755,156.919
C01778=1045.663,123.440,-88.955,170.538,36.753,156.919
C01779=1045.658,123.191,-88.934,170.535,36.752,156.919
C01780=1045.651,122.942,-88.914,170.533,36.750,156.919
C01781=1045.645,122.693,-88.894,170.532,36.749,156.918
C01782=1045.639,122.444,-88.872,170.530,36.747,156.918
C01783=1045.633,122.195,-88.852,170.528,36.746,156.918
C01784=1045.627,121.946,-88.832,170.525,36.744,156.917
C01785=1045.621,121.696,-88.811,170.524,36.743,156.917
